KUKA KRL program: MyProgram_302().src

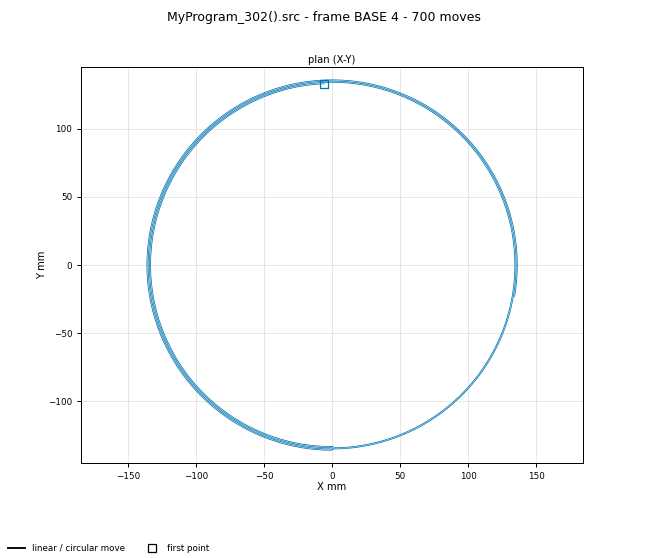
[picture p0: tool path of MyProgram_302().src in frame BASE 4, 700 of 700 moves have a stored position in this frame; points joined in program order, loops and branches not executed]
&ACCESS RVP
&REL 1
&PARAM TEMPLATE = C:\KRC\Roboter\Template\vorgabe
&PARAM EDITMASK = *
DEF MyProgram_302()
; ---- Setting reference (Base) ----
$BASE = BASE_DATA[4]

; --------------------------
; ---- Setting tool (TCP) ----
$TOOL = TOOL_DATA[3]
; --------------------------

$VEL.CP = VEL_APROX_PRINT
Startdeposition()
$VEL.CP = VEL_PRINT
LIN {X -5.8401,Y 133.2502,Z 180,A 93.9157,B 5.8389,C 0.0819,E1 5.8328,E2 358.4356} C_DIS
LIN {X -9.9087,Y 133.0081,Z 180,A 95.4392,B 5.8389,C 0.0849,E1 5.8286,E2 356.9401} C_DIS
LIN {X -13.164,Y 132.726,Z 180,A 96.8413,B 5.8389,C 0.0853,E1 5.8247,E2 355.5388} C_DIS
LIN {X -16.4317,Y 132.362,Z 180,A 98.2546,B 5.8389,C 0.0857,E1 5.8208,E2 354.1262} C_DIS
LIN {X -19.569,Y 131.9349,Z 180,A 99.6594,B 5.8389,C 0.0857,E1 5.8169,E2 352.7169} C_DIS
LIN {X -22.7973,Y 131.4155,Z 180,A 101.1451,B 5.8389,C 0.0853,E1 5.8128,E2 351.2223} C_DIS
LIN {X -26.0144,Y 130.8161,Z 180,A 102.4928,B 5.8389,C 0.0867,E1 5.8091,E2 349.8823} C_DIS
LIN {X -29.8878,Y 129.9846,Z 180,A 104.0027,B 5.8389,C 0.0899,E1 5.805,E2 348.3962} C_DIS
LIN {X -32.4071,Y 129.38,Z 180,A 105.3169,B 5.8389,C 0.0884,E1 5.8014,E2 347.0588} C_DIS
LIN {X -35.6706,Y 128.5181,Z 180,A 106.7192,B 5.8389,C 0.09,E1 5.7976,E2 345.663} C_DIS
LIN {X -39.0431,Y 127.5337,Z 180,A 108.1859,B 5.8388,C 0.0916,E1 5.7937,E2 344.2024} C_DIS
LIN {X -41.9497,Y 126.6076,Z 180,A 109.7012,B 5.8388,C 0.0904,E1 5.7896,E2 342.6636} C_DIS
LIN {X -46.4559,Y 125.0247,Z 180,A 111.6781,B 5.8388,C 0.0932,E1 5.7845,E2 340.697} C_DIS
LIN {X -49.6202,Y 123.8026,Z 180,A 113.0937,B 5.8388,C 0.0952,E1 5.7808,E2 339.2873} C_DIS
LIN {X -52.5449,Y 122.5903,Z 180,A 114.5896,B 5.8388,C 0.0952,E1 5.7769,E2 337.7762} C_DIS
LIN {X -55.543,Y 121.2616,Z 180,A 115.9158,B 5.8387,C 0.0977,E1 5.7736,E2 336.4609} C_DIS
LIN {X -58.4989,Y 119.864,Z 180,A 117.3346,B 5.8387,C 0.0992,E1 5.77,E2 335.0414} C_DIS
LIN {X -61.4202,Y 118.3941,Z 180,A 118.7379,B 5.8387,C 0.101,E1 5.7665,E2 333.6394} C_DIS
LIN {X -64.3234,Y 116.8431,Z 180,A 120.1855,B 5.8387,C 0.1026,E1 5.7629,E2 332.1889} C_DIS
LIN {X -67.1606,Y 115.2359,Z 180,A 121.6276,B 5.8386,C 0.1041,E1 5.7594,E2 330.743} C_DIS
LIN {X -69.9578,Y 113.5592,Z 180,A 123.0324,B 5.8386,C 0.1061,E1 5.7561,E2 329.3388} C_DIS
LIN {X -72.7953,Y 111.7614,Z 180,A 124.4937,B 5.8386,C 0.1081,E1 5.7527,E2 327.8763} C_DIS
LIN {X -75.4227,Y 110.0052,Z 180,A 125.8852,B 5.8385,C 0.1099,E1 5.7494,E2 326.4819} C_DIS
LIN {X -78.448,Y 107.8688,Z 180,A 127.5592,B 5.8385,C 0.1117,E1 5.7456,E2 324.7993} C_DIS
LIN {X -81.4564,Y 105.6156,Z 180,A 129.1159,B 5.8384,C 0.115,E1 5.7422,E2 323.2508} C_DIS
LIN {X -84.6152,Y 103.1022,Z 180,A 130.8894,B 5.8384,C 0.1177,E1 5.7383,E2 321.4741} C_DIS
LIN {X -87.1187,Y 100.9953,Z 180,A 132.463,B 5.8384,C 0.1186,E1 5.7349,E2 319.8816} C_DIS
LIN {X -90.2118,Y 98.2422,Z 180,A 134.2565,B 5.8382,C 0.1219,E1 5.7312,E2 318.0878} C_DIS
LIN {X -93.1509,Y 95.4606,Z 180,A 135.898,B 5.8382,C 0.1263,E1 5.7279,E2 316.4594} C_DIS
LIN {X -95.9962,Y 92.5986,Z 180,A 137.6763,B 5.8381,C 0.1293,E1 5.7245,E2 314.6773} C_DIS
LIN {X -98.8242,Y 89.574,Z 180,A 139.4792,B 5.838,C 0.1328,E1 5.721,E2 312.8731} C_DIS
LIN {X -101.5295,Y 86.4956,Z 180,A 141.4063,B 5.838,C 0.135,E1 5.7175,E2 310.9275} C_DIS
LIN {X -104.1336,Y 83.3429,Z 180,A 143.0495,B 5.8378,C 0.14,E1 5.7146,E2 309.2994} C_DIS
LIN {X -106.2103,Y 80.6799,Z 180,A 144.5409,B 5.8378,C 0.1428,E1 5.7121,E2 307.8044} C_DIS
LIN {X -108.0959,Y 78.1346,Z 180,A 145.9441,B 5.8377,C 0.1456,E1 5.7097,E2 306.3974} C_DIS
LIN {X -109.9841,Y 75.4533,Z 180,A 147.4489,B 5.8377,C 0.1479,E1 5.7073,E2 304.8823} C_DIS
LIN {X -111.8695,Y 72.6287,Z 180,A 148.8508,B 5.8375,C 0.152,E1 5.7052,E2 303.4885} C_DIS
LIN {X -113.5591,Y 69.9579,Z 180,A 150.2623,B 5.8375,C 0.1547,E1 5.7031,E2 302.0717} C_DIS
LIN {X -115.5146,Y 66.6793,Z 180,A 151.8127,B 5.8373,C 0.1596,E1 5.7009,E2 300.5336} C_DIS
LIN {X -116.8988,Y 64.2227,Z 180,A 153.1553,B 5.8373,C 0.1614,E1 5.6991,E2 299.1763} C_DIS
LIN {X -118.436,Y 61.3404,Z 180,A 154.5977,B 5.8372,C 0.1646,E1 5.6972,E2 297.7304} C_DIS
LIN {X -120.0778,Y 58.0592,Z 180,A 156.1261,B 5.8371,C 0.1691,E1 5.6953,E2 296.2091} C_DIS
LIN {X -121.3072,Y 55.4444,Z 180,A 157.4767,B 5.837,C 0.1713,E1 5.6937,E2 294.8465} C_DIS
LIN {X -122.9165,Y 51.7774,Z 180,A 159.3933,B 5.837,C 0.1739,E1 5.6916,E2 292.9078} C_DIS
LIN {X -124.4775,Y 47.9035,Z 180,A 161.1621,B 5.8368,C 0.179,E1 5.6898,E2 291.1436} C_DIS
LIN {X -126.0894,Y 43.4824,Z 180,A 163.1672,B 5.8366,C 0.1846,E1 5.6879,E2 289.1423} C_DIS
LIN {X -127.3112,Y 39.7702,Z 180,A 164.8428,B 5.8364,C 0.1892,E1 5.6865,E2 287.4686} C_DIS
LIN {X -128.0982,Y 37.151,Z 180,A 166.0629,B 5.8364,C 0.192,E1 5.6855,E2 286.244} C_DIS
LIN {X -128.9966,Y 33.9018,Z 180,A 167.5452,B 5.8362,C 0.1956,E1 5.6844,E2 284.7589} C_DIS
LIN {X -129.9243,Y 30.1519,Z 180,A 169.1106,B 5.8361,C 0.2011,E1 5.6834,E2 283.2062} C_DIS
LIN {X -130.5092,Y 27.5138,Z 180,A 170.4318,B 5.836,C 0.2029,E1 5.6826,E2 281.8666} C_DIS
LIN {X -131.1453,Y 24.3049,Z 180,A 171.8683,B 5.8359,C 0.2065,E1 5.6819,E2 280.4276} C_DIS
LIN {X -131.7018,Y 21.0799,Z 180,A 173.2973,B 5.8357,C 0.2103,E1 5.6812,E2 278.9969} C_DIS
LIN {X -132.1649,Y 17.947,Z 180,A 174.7293,B 5.8357,C 0.2135,E1 5.6807,E2 277.5573} C_DIS
LIN {X -132.5646,Y 14.7006,Z 180,A 176.1681,B 5.8355,C 0.2172,E1 5.6802,E2 276.1157} C_DIS
LIN {X -132.8853,Y 11.4385,Z 180,A 177.6287,B 5.8353,C 0.2207,E1 5.6798,E2 274.6498} C_DIS
LIN {X -133.1258,Y 8.1746,Z 180,A 179.0576,B 5.8353,C 0.2245,E1 5.6796,E2 273.2192} C_DIS
LIN {X -133.2866,Y 4.9068,Z 180,A -179.5165,B 5.8351,C 0.2283,E1 5.6794,E2 271.792} C_DIS
LIN {X -133.3749,Y 0.8313,Z 180,A -178.0632,B 5.8347,C 0.236,E1 5.6794,E2 270.3762} C_DIS
LIN {X -133.3679,Y -1.6325,Z 180,A -176.5813,B 5.8347,C 0.2352,E1 5.6794,E2 268.8437} C_DIS
LIN {X -133.2864,Y -4.9122,Z 180,A -175.1553,B 5.8347,C 0.239,E1 5.6794,E2 267.4167} C_DIS
LIN {X -133.1254,Y -8.1812,Z 180,A -173.7271,B 5.8345,C 0.2428,E1 5.6797,E2 265.9869} C_DIS
LIN {X -132.8762,Y -11.5458,Z 180,A -172.2661,B 5.8343,C 0.2468,E1 5.68,E2 264.5255} C_DIS
LIN {X -132.5536,Y -14.8028,Z 180,A -170.698,B 5.8342,C 0.2493,E1 5.6805,E2 262.9387} C_DIS
LIN {X -132.1502,Y -18.0593,Z 180,A -169.3858,B 5.834,C 0.2542,E1 5.681,E2 261.6395} C_DIS
LIN {X -131.6677,Y -21.2918,Z 180,A -167.9555,B 5.8338,C 0.2579,E1 5.6816,E2 260.2068} C_DIS
LIN {X -131.1247,Y -24.4125,Z 180,A -166.5253,B 5.8337,C 0.261,E1 5.6823,E2 258.7691} C_DIS
LIN {X -130.4641,Y -27.7227,Z 180,A -165.0366,B 5.8335,C 0.2647,E1 5.6831,E2 257.2766} C_DIS
LIN {X -129.7641,Y -30.8334,Z 180,A -163.6416,B 5.8334,C 0.2682,E1 5.684,E2 255.8794} C_DIS
LIN {X -128.9428,Y -34.1037,Z 180,A -162.1588,B 5.8332,C 0.2719,E1 5.6851,E2 254.3933} C_DIS
LIN {X -128.0976,Y -37.153,Z 180,A -160.7666,B 5.833,C 0.2753,E1 5.6861,E2 252.9979} C_DIS
LIN {X -127.1483,Y -40.2817,Z 180,A -159.3021,B 5.8329,C 0.2785,E1 5.6873,E2 251.5269} C_DIS
LIN {X -126.0624,Y -43.5603,Z 180,A -157.8574,B 5.8327,C 0.2829,E1 5.6886,E2 250.0879} C_DIS
LIN {X -125.0212,Y -46.4651,Z 180,A -156.4263,B 5.8326,C 0.2854,E1 5.69,E2 248.6445} C_DIS
LIN {X -123.5796,Y -50.1735,Z 180,A -154.8472,B 5.8323,C 0.2911,E1 5.6916,E2 247.0824} C_DIS
LIN {X -122.5879,Y -52.5505,Z 180,A -153.5732,B 5.8323,C 0.2924,E1 5.693,E2 245.7883} C_DIS
LIN {X -121.2627,Y -55.5407,Z 180,A -152.137,B 5.832,C 0.2957,E1 5.6947,E2 244.3491} C_DIS
LIN {X -119.838,Y -58.5516,Z 180,A -150.6937,B 5.8319,C 0.2992,E1 5.6964,E2 242.905} C_DIS
LIN {X -118.3945,Y -61.4194,Z 180,A -149.2856,B 5.8317,C 0.3023,E1 5.6982,E2 241.494} C_DIS
LIN {X -116.863,Y -64.2876,Z 180,A -147.8375,B 5.8315,C 0.3053,E1 5.7001,E2 240.0402} C_DIS
LIN {X -115.2646,Y -67.111,Z 180,A -146.2707,B 5.8315,C 0.307,E1 5.7024,E2 238.4526} C_DIS
LIN {X -113.5511,Y -69.9709,Z 180,A -144.9407,B 5.8312,C 0.3114,E1 5.7043,E2 237.136} C_DIS
LIN {X -111.7443,Y -72.8215,Z 180,A -143.4608,B 5.8311,C 0.3145,E1 5.7065,E2 235.6528} C_DIS
LIN {X -109.9836,Y -75.454,Z 180,A -142.0556,B 5.8309,C 0.3172,E1 5.7087,E2 234.2427} C_DIS
LIN {X -108.0943,Y -78.1368,Z 180,A -140.6414,B 5.8307,C 0.3204,E1 5.711,E2 232.8285} C_DIS
LIN {X -106.1145,Y -80.8053,Z 180,A -139.1884,B 5.8306,C 0.3233,E1 5.7135,E2 231.3728} C_DIS
LIN {X -103.6547,Y -83.9373,Z 180,A -137.4174,B 5.8304,C 0.3264,E1 5.7166,E2 229.5948} C_DIS
LIN {X -100.9949,Y -87.1191,Z 180,A -135.4726,B 5.8303,C 0.3284,E1 5.7201,E2 227.6303} C_DIS
LIN {X -98.237,Y -90.2175,Z 180,A -133.676,B 5.8301,C 0.3319,E1 5.7235,E2 225.8323} C_DIS
LIN {X -95.4637,Y -93.1478,Z 180,A -132.0371,B 5.8298,C 0.3364,E1 5.7266,E2 224.2056} C_DIS
LIN {X -92.6027,Y -95.9922,Z 180,A -130.2614,B 5.8297,C 0.3393,E1 5.7302,E2 222.4249} C_DIS
LIN {X -89.5801,Y -98.8186,Z 180,A -128.4607,B 5.8295,C 0.3423,E1 5.7339,E2 220.6216} C_DIS
LIN {X -86.4961,Y -101.529,Z 180,A -126.5401,B 5.8295,C 0.3438,E1 5.738,E2 218.6818} C_DIS
LIN {X -83.3456,Y -104.1314,Z 180,A -124.8384,B 5.8292,C 0.3474,E1 5.7417,E2 216.987} C_DIS
LIN {X -80.6705,Y -106.2174,Z 180,A -123.4167,B 5.829,C 0.3502,E1 5.7448,E2 215.5699} C_DIS
LIN {X -78.1287,Y -108.1002,Z 180,A -122.0232,B 5.829,C 0.352,E1 5.7479,E2 214.1722} C_DIS
LIN {X -75.4533,Y -109.9841,Z 180,A -120.618,B 5.8288,C 0.3541,E1 5.7512,E2 212.7671} C_DIS
LIN {X -72.6468,Y -111.8578,Z 180,A -119.1506,B 5.8287,C 0.3561,E1 5.7546,E2 211.2976} C_DIS
LIN {X -69.971,Y -113.551,Z 180,A -117.7497,B 5.8286,C 0.3575,E1 5.7579,E2 209.8917} C_DIS
LIN {X -67.0769,Y -115.2843,Z 180,A -116.2249,B 5.8286,C 0.3586,E1 5.7616,E2 208.3573} C_DIS
LIN {X -63.6192,Y -117.228,Z 180,A -114.6815,B 5.8283,C 0.3626,E1 5.7653,E2 206.834} C_DIS
LIN {X -61.3282,Y -118.4424,Z 180,A -113.4475,B 5.8283,C 0.3626,E1 5.7684,E2 205.5849} C_DIS
LIN {X -58.4051,Y -119.9102,Z 180,A -112.0301,B 5.8282,C 0.3641,E1 5.772,E2 204.1659} C_DIS
LIN {X -55.4488,Y -121.3052,Z 180,A -110.6141,B 5.8281,C 0.3655,E1 5.7756,E2 202.7482} C_DIS
LIN {X -52.4577,Y -122.6281,Z 180,A -109.206,B 5.8281,C 0.3669,E1 5.7792,E2 201.3396} C_DIS
LIN {X -49.5299,Y -123.839,Z 180,A -107.8163,B 5.8279,C 0.3679,E1 5.7828,E2 199.946} C_DIS
LIN {X -46.3584,Y -125.0612,Z 180,A -106.3358,B 5.8279,C 0.369,E1 5.7867,E2 198.4628} C_DIS
LIN {X -43.3991,Y -126.1182,Z 180,A -104.9873,B 5.8279,C 0.3701,E1 5.7902,E2 197.1142} C_DIS
LIN {X -40.2328,Y -127.1639,Z 180,A -103.5591,B 5.8277,C 0.3713,E1 5.794,E2 195.6862} C_DIS
LIN {X -37.2598,Y -128.0663,Z 180,A -102.1668,B 5.8277,C 0.3715,E1 5.7978,E2 194.2864} C_DIS
LIN {X -33.7056,Y -129.0489,Z 180,A -100.63,B 5.8277,C 0.3731,E1 5.8019,E2 192.7552} C_DIS
LIN {X -30.8137,Y -129.7689,Z 180,A -99.337,B 5.8276,C 0.3736,E1 5.8054,E2 191.4602} C_DIS
LIN {X -27.5186,Y -130.5082,Z 180,A -97.8837,B 5.8276,C 0.3743,E1 5.8094,E2 190.0062} C_DIS
LIN {X -24.3131,Y -131.1437,Z 180,A -96.3211,B 5.8276,C 0.3729,E1 5.8137,E2 188.4231} C_DIS
LIN {X -21.0911,Y -131.7001,Z 180,A -95.0816,B 5.8275,C 0.3754,E1 5.8171,E2 187.2041} C_DIS
LIN {X -17.958,Y -132.1635,Z 180,A -93.6817,B 5.8275,C 0.3754,E1 5.821,E2 185.7987} C_DIS
LIN {X -14.6983,Y -132.5648,Z 180,A -92.2718,B 5.8275,C 0.3756,E1 5.8249,E2 184.3883} C_DIS
LIN {X -11.4444,Y -132.8848,Z 180,A -90.8248,B 5.8275,C 0.3753,E1 5.8289,E2 182.9354} C_DIS
LIN {X -8.1833,Y -133.1253,Z 180,A -89.4562,B 5.8275,C 0.3758,E1 5.8327,E2 181.5708} C_DIS
LIN {X -4.9184,Y -133.2862,Z 180,A -88.0669,B 5.8275,C 0.376,E1 5.8366,E2 180.1828} C_DIS
LIN {X -1.6521,Y -133.3676,Z 180,A -86.6466,B 5.8275,C 0.3757,E1 5.8406,E2 178.7597} C_DIS
LIN {X 0.9654,Y -133.3724,Z 180,A -85.8773,B 5.8272,C 0.3801,E1 5.8426,E2 178.0345} C_DIS
Enddeposition()
LIN {X 0.9654,Y -133.3724,Z 180,A -85.8773,B 5.8272,C 0.3801,E1 5.8426,E2 178.0345} C_DIS
Startdeposition()
$VEL.CP = VEL_PRINT
LIN {X -1.8229,Y -134.2676,Z 180,A -87.4081,B 5.8265,C 0.3879,E1 5.838,E2 179.6414} C_DIS
LIN {X -5.9362,Y -134.1498,Z 180,A -89.2358,B 5.8265,C 0.3889,E1 5.8329,E2 181.479} C_DIS
LIN {X -10.4243,Y -133.8756,Z 180,A -90.9726,B 5.8266,C 0.3865,E1 5.8281,E2 183.1938} C_DIS
LIN {X -13.6518,Y -133.5853,Z 180,A -92.7112,B 5.8264,C 0.3907,E1 5.8232,E2 184.9776} C_DIS
LIN {X -16.9255,Y -133.2092,Z 180,A -93.6954,B 5.8267,C 0.3851,E1 5.8206,E2 185.9093} C_DIS
LIN {X -19.5444,Y -132.8503,Z 180,A -94.891,B 5.8267,C 0.3857,E1 5.8173,E2 187.1138} C_DIS
LIN {X -23.1124,Y -132.2762,Z 180,A -96.6307,B 5.8266,C 0.3876,E1 5.8124,E2 188.8789} C_DIS
LIN {X -27.0527,Y -131.526,Z 180,A -98.1959,B 5.8267,C 0.385,E1 5.8081,E2 190.4262} C_DIS
LIN {X -30.9558,Y -130.6631,Z 180,A -100.0353,B 5.8267,C 0.3858,E1 5.8031,E2 192.283} C_DIS
LIN {X -35.3302,Y -129.5499,Z 180,A -102.2882,B 5.8265,C 0.3885,E1 5.7969,E2 194.5771} C_DIS
LIN {X -39.0512,Y -128.4753,Z 180,A -103.9879,B 5.8265,C 0.3878,E1 5.7923,E2 196.283} C_DIS
LIN {X -43.1127,Y -127.171,Z 180,A -105.3156,B 5.827,C 0.3806,E1 5.789,E2 197.5496} C_DIS
LIN {X -46.1895,Y -126.0865,Z 180,A -107.0216,B 5.8269,C 0.3831,E1 5.7844,E2 199.2952} C_DIS
LIN {X -51.1313,Y -124.1645,Z 180,A -108.9572,B 5.8273,C 0.3772,E1 5.7795,E2 201.1902} C_DIS
LIN {X -53.5217,Y -123.1514,Z 180,A -110.1581,B 5.8273,C 0.3772,E1 5.7764,E2 202.4028} C_DIS
LIN {X -57.232,Y -121.4734,Z 180,A -111.8503,B 5.8274,C 0.3747,E1 5.7721,E2 204.0896} C_DIS
LIN {X -59.6757,Y -120.29,Z 180,A -113.1398,B 5.8274,C 0.3749,E1 5.7688,E2 205.3955} C_DIS
LIN {X -63.8676,Y -118.1202,Z 180,A -115.1667,B 5.8275,C 0.3725,E1 5.7638,E2 207.4242} C_DIS
LIN {X -67.6152,Y -116.0158,Z 180,A -117.0786,B 5.8276,C 0.371,E1 5.7591,E2 209.3458} C_DIS
LIN {X -70.8161,Y -114.0895,Z 180,A -118.5521,B 5.8279,C 0.3674,E1 5.7557,E2 210.8042} C_DIS
LIN {X -73.4828,Y -112.3912,Z 180,A -120.0772,B 5.8279,C 0.3674,E1 5.752,E2 212.3513} C_DIS
LIN {X -76.8332,Y -110.1272,Z 180,A -121.8054,B 5.828,C 0.3648,E1 5.7481,E2 214.0797} C_DIS
LIN {X -80.357,Y -107.583,Z 180,A -123.6442,B 5.8282,C 0.3617,E1 5.7439,E2 215.9164} C_DIS
LIN {X -83.8659,Y -104.871,Z 180,A -125.5135,B 5.8284,C 0.3583,E1 5.7398,E2 217.7826} C_DIS
LIN {X -86.7787,Y -102.4735,Z 180,A -127.2167,B 5.8286,C 0.3565,E1 5.7361,E2 219.4972} C_DIS
LIN {X -90.0905,Y -99.5744,Z 180,A -129.1455,B 5.8287,C 0.3536,E1 5.7321,E2 221.4319} C_DIS
LIN {X -93.5149,Y -96.3655,Z 180,A -131.098,B 5.829,C 0.3493,E1 5.7282,E2 223.3779} C_DIS
LIN {X -96.2125,Y -93.6729,Z 180,A -132.7735,B 5.8291,C 0.3466,E1 5.7249,E2 225.0592} C_DIS
LIN {X -98.7892,Y -90.9507,Z 180,A -134.4306,B 5.8293,C 0.344,E1 5.7217,E2 226.7229} C_DIS
LIN {X -101.2522,Y -88.2004,Z 180,A -136.0603,B 5.8295,C 0.3413,E1 5.7187,E2 228.359} C_DIS
LIN {X -104.2235,Y -84.6695,Z 180,A -138.0297,B 5.8297,C 0.3371,E1 5.7152,E2 230.3278} C_DIS
LIN {X -106.5852,Y -81.6757,Z 180,A -139.6703,B 5.8299,C 0.3336,E1 5.7124,E2 231.9695} C_DIS
LIN {X -109.0027,Y -78.4212,Z 180,A -141.522,B 5.83,C 0.331,E1 5.7093,E2 233.8356} C_DIS
LIN {X -111.7464,Y -74.4585,Z 180,A -143.4191,B 5.8304,C 0.3246,E1 5.7063,E2 235.7122} C_DIS
LIN {X -113.3521,Y -71.9914,Z 180,A -144.7748,B 5.8305,C 0.3227,E1 5.7043,E2 237.0798} C_DIS
LIN {X -115.3599,Y -68.7271,Z 180,A -147.8317,B 5.83,C 0.3326,E1 5.6997,E2 240.3093} C_DIS
LIN {X -119.6052,Y -61.0359,Z 180,A -149.9919,B 5.8313,C 0.3079,E1 5.6971,E2 242.274} C_DIS
LIN {X -121.4935,Y -57.19,Z 180,A -152.1421,B 5.8313,C 0.3064,E1 5.6944,E2 244.4631} C_DIS
LIN {X -122.6668,Y -54.6231,Z 180,A -153.3886,B 5.8315,C 0.3037,E1 5.693,E2 245.714} C_DIS
LIN {X -124.129,Y -51.2163,Z 180,A -154.9876,B 5.8317,C 0.2998,E1 5.6913,E2 247.3143} C_DIS
LIN {X -125.6383,Y -47.391,Z 180,A -156.5791,B 5.832,C 0.2936,E1 5.6897,E2 248.8847} C_DIS
LIN {X -126.422,Y -45.2589,Z 180,A -157.8208,B 5.832,C 0.2936,E1 5.6885,E2 250.1594} C_DIS
LIN {X -127.5238,Y -42.0553,Z 180,A -159.2082,B 5.8323,C 0.2892,E1 5.6872,E2 251.5388} C_DIS
LIN {X -128.5924,Y -38.6682,Z 180,A -160.7647,B 5.8324,C 0.2855,E1 5.6859,E2 253.0994} C_DIS
LIN {X -129.5062,Y -35.489,Z 180,A -162.3212,B 5.8326,C 0.283,E1 5.6848,E2 254.6729} C_DIS
LIN {X -130.9359,Y -29.7766,Z 180,A -164.7998,B 5.8329,C 0.2758,E1 5.6831,E2 257.1456} C_DIS
LIN {X -131.6865,Y -26.2638,Z 180,A -166.4132,B 5.8331,C 0.2723,E1 5.6822,E2 258.7678} C_DIS
LIN {X -132.284,Y -23.0684,Z 180,A -167.924,B 5.8331,C 0.2696,E1 5.6814,E2 260.2928} C_DIS
LIN {X -132.9526,Y -18.8284,Z 180,A -169.7276,B 5.8334,C 0.2642,E1 5.6807,E2 262.0917} C_DIS
LIN {X -133.4808,Y -14.6235,Z 180,A -171.5757,B 5.8337,C 0.2594,E1 5.6801,E2 263.9434} C_DIS
LIN {X -133.877,Y -10.4048,Z 180,A -173.3775,B 5.8339,C 0.2542,E1 5.6796,E2 265.7431} C_DIS
LIN {X -134.0726,Y -7.4837,Z 180,A -174.8802,B 5.8339,C 0.253,E1 5.6794,E2 267.2757} C_DIS
LIN {X -134.2477,Y -3.004,Z 180,A -176.7939,B 5.8342,C 0.2476,E1 5.6792,E2 269.188} C_DIS
LIN {X -134.2747,Y 1.2521,Z 180,A -178.5999,B 5.8344,C 0.2423,E1 5.6792,E2 270.9914} C_DIS
LIN {X -134.1737,Y 5.3251,Z 180,A 179.6874,B 5.8346,C 0.2371,E1 5.6794,E2 272.6995} C_DIS
LIN {X -134.0112,Y 8.4826,Z 180,A 178.3108,B 5.8347,C 0.2335,E1 5.6796,E2 274.0783} C_DIS
LIN {X -133.7853,Y 11.5076,Z 180,A 176.9868,B 5.8349,C 0.2301,E1 5.6799,E2 275.4049} C_DIS
LIN {X -133.4736,Y 14.6901,Z 180,A 175.5902,B 5.835,C 0.2265,E1 5.6803,E2 276.8043} C_DIS
LIN {X -133.0711,Y 17.9794,Z 180,A 173.9883,B 5.8351,C 0.2242,E1 5.6809,E2 278.4277} C_DIS
LIN {X -132.3686,Y 22.5758,Z 180,A 171.9674,B 5.8353,C 0.219,E1 5.6818,E2 280.4514} C_DIS
LIN {X -131.5306,Y 27.0302,Z 180,A 170.0654,B 5.8355,C 0.2133,E1 5.6828,E2 282.3479} C_DIS
LIN {X -130.446,Y 31.8568,Z 180,A 168.0066,B 5.8358,C 0.2069,E1 5.6841,E2 284.3986} C_DIS
LIN {X -129.6981,Y 34.7746,Z 180,A 166.5489,B 5.8358,C 0.2049,E1 5.6851,E2 285.876} C_DIS
LIN {X -128.7451,Y 38.154,Z 180,A 165.087,B 5.836,C 0.2005,E1 5.6863,E2 287.3322} C_DIS
LIN {X -127.7191,Y 41.4613,Z 180,A 163.6201,B 5.8361,C 0.1964,E1 5.6875,E2 288.7965} C_DIS
LIN {X -126.7327,Y 44.3825,Z 180,A 162.1143,B 5.8361,C 0.1946,E1 5.6889,E2 290.324} C_DIS
LIN {X -125.4252,Y 47.9571,Z 180,A 160.6153,B 5.8364,C 0.1891,E1 5.6904,E2 291.8066} C_DIS
LIN {X -124.4052,Y 50.5399,Z 180,A 159.3751,B 5.8364,C 0.1864,E1 5.6917,E2 293.0524} C_DIS
LIN {X -123.0342,Y 53.7929,Z 180,A 157.8355,B 5.8366,C 0.1828,E1 5.6933,E2 294.5946} C_DIS
LIN {X -121.6853,Y 56.7774,Z 180,A 156.378,B 5.8366,C 0.1797,E1 5.6951,E2 296.0582} C_DIS
LIN {X -119.6414,Y 60.9648,Z 180,A 154.5514,B 5.8368,C 0.1731,E1 5.6973,E2 297.8635} C_DIS
LIN {X -118.1614,Y 63.7909,Z 180,A 152.8627,B 5.8368,C 0.1728,E1 5.6995,E2 299.5904} C_DIS
LIN {X -116.0354,Y 67.5813,Z 180,A 150.9864,B 5.837,C 0.1684,E1 5.7021,E2 301.4677} C_DIS
LIN {X -114.1029,Y 70.7946,Z 180,A 148.9129,B 5.837,C 0.169,E1 5.7053,E2 303.596} C_DIS
LIN {X -111.7453,Y 74.4602,Z 180,A 147.4305,B 5.8372,C 0.1609,E1 5.7075,E2 305.0319} C_DIS
LIN {X -109.0975,Y 78.2886,Z 180,A 145.4013,B 5.8373,C 0.1567,E1 5.7107,E2 307.0645} C_DIS
LIN {X -106.8983,Y 81.2663,Z 180,A 143.8891,B 5.8374,C 0.1525,E1 5.7133,E2 308.5674} C_DIS
LIN {X -104.445,Y 84.3954,Z 180,A 142.0516,B 5.8374,C 0.1501,E1 5.7165,E2 310.4202} C_DIS
LIN {X -101.5169,Y 87.8963,Z 180,A 140.0565,B 5.8376,C 0.1463,E1 5.7201,E2 312.4191} C_DIS
LIN {X -98.5584,Y 91.2016,Z 180,A 138.1918,B 5.8376,C 0.142,E1 5.7236,E2 314.2789} C_DIS
LIN {X -95.7512,Y 94.1437,Z 180,A 136.3912,B 5.8378,C 0.1391,E1 5.7271,E2 316.0858} C_DIS
LIN {X -92.5547,Y 97.2884,Z 180,A 134.4713,B 5.8378,C 0.1354,E1 5.7309,E2 318.0048} C_DIS
LIN {X -89.2963,Y 100.2877,Z 180,A 132.5062,B 5.8379,C 0.1326,E1 5.735,E2 319.9773} C_DIS
LIN {X -85.941,Y 103.1776,Z 180,A 130.5766,B 5.8379,C 0.1295,E1 5.7391,E2 321.91} C_DIS
LIN {X -82.5668,Y 105.8971,Z 180,A 128.6761,B 5.838,C 0.1268,E1 5.7433,E2 323.8152} C_DIS
LIN {X -78.9123,Y 108.6471,Z 180,A 126.7683,B 5.8381,C 0.123,E1 5.7476,E2 325.7162} C_DIS
LIN {X -73.5343,Y 112.3573,Z 180,A 123.6484,B 5.8381,C 0.1221,E1 5.7549,E2 328.8731} C_DIS
LIN {X -70.5442,Y 114.2584,Z 180,A 122.6292,B 5.8383,C 0.1147,E1 5.7572,E2 329.8328} C_DIS
LIN {X -68.0549,Y 115.7577,Z 180,A 121.1966,B 5.8383,C 0.1149,E1 5.7607,E2 331.2873} C_DIS
LIN {X -63.1842,Y 118.4874,Z 180,A 118.804,B 5.8383,C 0.1118,E1 5.7665,E2 333.6794} C_DIS
LIN {X -59.0297,Y 120.6086,Z 180,A 116.7474,B 5.8383,C 0.11,E1 5.7717,E2 335.7422} C_DIS
LIN {X -56.1305,Y 121.9844,Z 180,A 115.4098,B 5.8384,C 0.108,E1 5.775,E2 337.0751} C_DIS
LIN {X -52.8449,Y 123.4441,Z 180,A 113.7464,B 5.8384,C 0.1077,E1 5.7793,E2 338.7528} C_DIS
LIN {X -49.6878,Y 124.7486,Z 180,A 111.4479,B 5.8383,C 0.1154,E1 5.7856,E2 341.1489} C_DIS
LIN {X -43.5256,Y 127.0298,Z 180,A 109.5502,B 5.8385,C 0.1028,E1 5.7903,E2 342.9385} C_DIS
LIN {X -38.0339,Y 128.7802,Z 180,A 107.2884,B 5.8385,C 0.0986,E1 5.7962,E2 345.1752} C_DIS
LIN {X -35.2972,Y 129.5587,Z 180,A 105.9102,B 5.8385,C 0.0995,E1 5.8,E2 346.5723} C_DIS
LIN {X -32.4186,Y 130.3084,Z 180,A 104.6358,B 5.8385,C 0.0987,E1 5.8034,E2 347.8465} C_DIS
LIN {X -29.6954,Y 130.9545,Z 180,A 103.3822,B 5.8385,C 0.0987,E1 5.8069,E2 349.1063} C_DIS
LIN {X -25.9469,Y 131.7504,Z 180,A 101.7804,B 5.8385,C 0.0974,E1 5.8112,E2 350.7033} C_DIS
LIN {X -22.9099,Y 132.3123,Z 180,A 100.292,B 5.8385,C 0.0988,E1 5.8154,E2 352.2111} C_DIS
LIN {X -18.4899,Y 133.001,Z 180,A 98.5148,B 5.8386,C 0.0965,E1 5.8202,E2 353.9718} C_DIS
LIN {X -13.0322,Y 133.6454,Z 180,A 96.3422,B 5.8386,C 0.0938,E1 5.8262,E2 356.1226} C_DIS
LIN {X -9.7194,Y 133.927,Z 180,A 94.6822,B 5.8386,C 0.0964,E1 5.8309,E2 357.8105} C_DIS
LIN {X -6.088,Y 134.1428,Z 180,A 93.0193,B 5.8386,C 0.0975,E1 5.8356,E2 359.4859} C_DIS
LIN {X -2.467,Y 134.2569,Z 180,A 91.5934,B 5.8386,C 0.096,E1 5.8395,E2 360.8969} C_DIS
LIN {X 1.1007,Y 134.2753,Z 180,A 90.1887,B 5.8386,C 0.0946,E1 5.8434,E2 362.2869} C_DIS
LIN {X 4.6564,Y 134.1998,Z 180,A 88.6949,B 5.8386,C 0.0945,E1 5.8476,E2 363.7774} C_DIS
LIN {X 7.3307,Y 134.0803,Z 180,A 87.2919,B 5.8386,C 0.0979,E1 5.8516,E2 365.2108} C_DIS
LIN {X 10.9211,Y 133.8349,Z 180,A 85.7758,B 5.8386,C 0.098,E1 5.8558,E2 366.724} C_DIS
LIN {X 14.8909,Y 133.452,Z 180,A 84.23,B 5.8386,C 0.0967,E1 5.86,E2 368.2507} C_DIS
LIN {X 18.887,Y 132.9442,Z 180,A 82.568,B 5.8386,C 0.0967,E1 5.8646,E2 369.9053} C_DIS
LIN {X 22.3354,Y 132.4087,Z 180,A 81.0552,B 5.8386,C 0.0977,E1 5.8688,E2 371.4205} C_DIS
LIN {X 25.9928,Y 131.7416,Z 180,A 79.3333,B 5.8386,C 0.1003,E1 5.8736,E2 373.1581} C_DIS
LIN {X 30.1267,Y 130.8559,Z 180,A 77.6008,B 5.8386,C 0.1005,E1 5.8783,E2 374.8816} C_DIS
LIN {X 35.9171,Y 129.3865,Z 180,A 74.6568,B 5.8384,C 0.1076,E1 5.8863,E2 377.8718} C_DIS
LIN {X 39.9713,Y 128.1932,Z 180,A 73.3449,B 5.8385,C 0.1027,E1 5.8897,E2 379.1251} C_DIS
LIN {X 43.235,Y 127.1305,Z 180,A 71.6493,B 5.8385,C 0.1071,E1 5.8942,E2 380.848} C_DIS
LIN {X 47.3091,Y 125.669,Z 180,A 69.9995,B 5.8385,C 0.1064,E1 5.8985,E2 382.4739} C_DIS
LIN {X 50.6514,Y 124.3602,Z 180,A 68.5478,B 5.8385,C 0.107,E1 5.9022,E2 383.916} C_DIS
LIN {X 53.9842,Y 122.9515,Z 180,A 67.0057,B 5.8384,C 0.1087,E1 5.9062,E2 385.4578} C_DIS
LIN {X 56.7098,Y 121.7166,Z 180,A 65.7474,B 5.8384,C 0.11,E1 5.9094,E2 386.7137} C_DIS
LIN {X 59.7538,Y 120.2514,Z 180,A 64.2889,B 5.8384,C 0.1121,E1 5.9131,E2 388.1741} C_DIS
LIN {X 63.6861,Y 118.2177,Z 180,A 62.356,B 5.8383,C 0.1152,E1 5.9178,E2 390.1123} C_DIS
LIN {X 67.593,Y 116.0286,Z 180,A 60.5146,B 5.8383,C 0.117,E1 5.9223,E2 391.9454} C_DIS
LIN {X 70.7099,Y 114.1556,Z 180,A 59.0352,B 5.8383,C 0.1184,E1 5.9258,E2 393.4163} C_DIS
LIN {X 73.8141,Y 112.1731,Z 180,A 57.4868,B 5.8382,C 0.1205,E1 5.9294,E2 394.9618} C_DIS
LIN {X 76.9618,Y 110.0377,Z 180,A 55.7717,B 5.8381,C 0.1244,E1 5.9334,E2 396.6881} C_DIS
LIN {X 80.1819,Y 107.7134,Z 180,A 54.1128,B 5.8381,C 0.1268,E1 5.9371,E2 398.3429} C_DIS
LIN {X 83.8198,Y 104.9076,Z 180,A 52.2256,B 5.838,C 0.1293,E1 5.9413,E2 400.2217} C_DIS
LIN {X 86.605,Y 102.6208,Z 180,A 50.6696,B 5.838,C 0.1323,E1 5.9446,E2 401.7801} C_DIS
LIN {X 90.4223,Y 99.2733,Z 180,A 48.7849,B 5.838,C 0.1324,E1 5.9485,E2 403.6314} C_DIS
LIN {X 92.5684,Y 97.2754,Z 180,A 47.3214,B 5.8378,C 0.1379,E1 5.9515,E2 405.1207} C_DIS
LIN {X 95.577,Y 94.3214,Z 180,A 45.5045,B 5.8377,C 0.1418,E1 5.9551,E2 406.9401} C_DIS
LIN {X 98.0657,Y 91.7307,Z 180,A 44.0118,B 5.8377,C 0.1445,E1 5.9579,E2 408.4283} C_DIS
LIN {X 101.1335,Y 88.3364,Z 180,A 42.1376,B 5.8375,C 0.1475,E1 5.9614,E2 410.2937} C_DIS
LIN {X 103.996,Y 84.9479,Z 180,A 40.2576,B 5.8375,C 0.1515,E1 5.9648,E2 412.1728} C_DIS
LIN {X 106.8095,Y 81.3825,Z 180,A 38.4037,B 5.8374,C 0.1546,E1 5.9679,E2 414.0172} C_DIS
LIN {X 109.4242,Y 77.8316,Z 180,A 36.5302,B 5.8373,C 0.1588,E1 5.971,E2 415.8904} C_DIS
LIN {X 111.8797,Y 74.2589,Z 180,A 34.6686,B 5.8371,C 0.1634,E1 5.9739,E2 417.7542} C_DIS
LIN {X 114.0626,Y 70.8594,Z 180,A 33.0981,B 5.8371,C 0.1652,E1 5.9762,E2 419.3068} C_DIS
LIN {X 116.1136,Y 67.4462,Z 180,A 31.3436,B 5.8369,C 0.1702,E1 5.9787,E2 421.0688} C_DIS
LIN {X 118.309,Y 63.5162,Z 180,A 29.3918,B 5.8368,C 0.1755,E1 5.9814,E2 423.0253} C_DIS
LIN {X 120.4073,Y 59.4379,Z 180,A 27.5615,B 5.8367,C 0.1786,E1 5.9836,E2 424.8411} C_DIS
LIN {X 122.1459,Y 55.7813,Z 180,A 25.9847,B 5.8367,C 0.1807,E1 5.9855,E2 426.4005} C_DIS
LIN {X 123.2458,Y 53.3035,Z 180,A 24.4653,B 5.8363,C 0.1893,E1 5.9872,E2 427.9644} C_DIS
LIN {X 124.6709,Y 49.8805,Z 180,A 22.7558,B 5.8361,C 0.1954,E1 5.989,E2 429.6902} C_DIS
LIN {X 126.2827,Y 45.6454,Z 180,A 21.2942,B 5.8362,C 0.1934,E1 5.9904,E2 431.0958} C_DIS
LIN {X 128.0814,Y 40.3271,Z 180,A 19.0623,B 5.8361,C 0.1974,E1 5.9923,E2 433.3092} C_DIS
LIN {X 129.2445,Y 36.4247,Z 180,A 17.3443,B 5.8359,C 0.2018,E1 5.9936,E2 435.0259} C_DIS
LIN {X 130.2613,Y 32.604,Z 180,A 15.5872,B 5.8357,C 0.2075,E1 5.9949,E2 436.7927} C_DIS
LIN {X 131.3604,Y 27.8488,Z 180,A 13.6961,B 5.8357,C 0.2104,E1 5.996,E2 438.6617} C_DIS
LIN {X 132.0168,Y 24.5537,Z 180,A 12.2804,B 5.8355,C 0.2141,E1 5.9968,E2 440.0762} C_DIS
LIN {X 132.6829,Y 20.6428,Z 180,A 10.6122,B 5.8353,C 0.2185,E1 5.9975,E2 441.7425} C_DIS
LIN {X 133.2533,Y 16.5799,Z 180,A 8.9812,B 5.8353,C 0.2216,E1 5.9981,E2 443.3602} C_DIS
LIN {X 133.5382,Y 14.0897,Z 180,A 7.943,B 5.8351,C 0.2241,E1 5.9984,E2 444.3953} C_DIS
LIN {X 133.7815,Y 11.5538,Z 180,A 6.9204,B 5.8351,C 0.2262,E1 5.9987,E2 445.4108} C_DIS
LIN {X 133.9836,Y 8.9309,Z 180,A 5.7832,B 5.8349,C 0.2296,E1 5.9989,E2 446.5507} C_DIS
LIN {X 134.1437,Y 6.0686,Z 180,A 4.3933,B 5.8347,C 0.2357,E1 5.9991,E2 447.962} C_DIS
LIN {X 134.2708,Y 1.6275,Z 180,A 2.7791,B 5.8347,C 0.2367,E1 5.9992,E2 449.543} C_DIS
LIN {X 134.278,Y -0.7661,Z 180,A 1.5874,B 5.8344,C 0.2423,E1 5.9992,E2 450.7565} C_DIS
LIN {X 134.1797,Y -5.1715,Z 180,A -0.2,B 5.8342,C 0.2462,E1 5.9991,E2 452.5339} C_DIS
LIN {X 133.9953,Y -8.7404,Z 180,A -1.7823,B 5.834,C 0.2515,E1 5.9988,E2 454.1246} C_DIS
LIN {X 133.7002,Y -12.4622,Z 180,A -3.0901,B 5.834,C 0.2515,E1 5.9985,E2 455.3985} C_DIS
LIN {X 133.4347,Y -15.0517,Z 180,A -4.2486,B 5.8338,C 0.2555,E1 5.9981,E2 456.5638} C_DIS
LIN {X 133.1148,Y -17.6456,Z 180,A -5.3021,B 5.8338,C 0.2577,E1 5.9978,E2 457.6105} C_DIS
LIN {X 132.7618,Y -20.1331,Z 180,A -6.3337,B 5.8336,C 0.2601,E1 5.9973,E2 458.6381} C_DIS
LIN {X 132.1676,Y -23.719,Z 180,A -8.0262,B 5.8333,C 0.2667,E1 5.9965,E2 460.3494} C_DIS
LIN {X 131.4342,Y -27.504,Z 180,A -9.5034,B 5.8333,C 0.2687,E1 5.9957,E2 461.8073} C_DIS
LIN {X 130.809,Y -30.3322,Z 180,A -10.7,B 5.8331,C 0.2715,E1 5.995,E2 463.0001} C_DIS
LIN {X 129.9833,Y -33.6994,Z 180,A -12.5818,B 5.8326,C 0.2819,E1 5.9937,E2 464.933} C_DIS
LIN {X 128.9879,Y -37.3245,Z 180,A -13.5942,B 5.8328,C 0.2772,E1 5.993,E2 465.8736} C_DIS
LIN {X 128.1469,Y -40.1223,Z 180,A -15.2321,B 5.8324,C 0.2867,E1 5.9916,E2 467.5611} C_DIS
LIN {X 126.787,Y -44.226,Z 180,A -16.7826,B 5.8324,C 0.2871,E1 5.9902,E2 469.0767} C_DIS
LIN {X 125.5875,Y -47.5267,Z 180,A -18.2485,B 5.8322,C 0.2907,E1 5.9888,E2 470.54} C_DIS
LIN {X 124.3801,Y -50.6021,Z 180,A -19.7542,B 5.8319,C 0.2959,E1 5.9872,E2 472.0588} C_DIS
LIN {X 122.8993,Y -54.1033,Z 180,A -21.1764,B 5.8319,C 0.2971,E1 5.9856,E2 473.4577} C_DIS
LIN {X 121.7994,Y -56.5308,Z 180,A -22.4118,B 5.8316,C 0.3016,E1 5.9842,E2 474.7063} C_DIS
LIN {X 120.1974,Y -59.8633,Z 180,A -23.9141,B 5.8315,C 0.3046,E1 5.9823,E2 476.2008} C_DIS
LIN {X 117.7723,Y -64.5063,Z 180,A -26.0771,B 5.8312,C 0.3092,E1 5.9795,E2 478.3568} C_DIS
LIN {X 115.7201,Y -68.119,Z 180,A -27.8288,B 5.831,C 0.3133,E1 5.9771,E2 480.1075} C_DIS
LIN {X 113.4985,Y -71.7594,Z 180,A -29.6084,B 5.8308,C 0.3172,E1 5.9745,E2 481.8837} C_DIS
LIN {X 111.089,Y -75.4359,Z 180,A -31.4124,B 5.8306,C 0.3207,E1 5.9717,E2 483.6805} C_DIS
LIN {X 108.7347,Y -78.7914,Z 180,A -33.1894,B 5.8304,C 0.3253,E1 5.9688,E2 485.4626} C_DIS
LIN {X 106.2386,Y -82.1262,Z 180,A -34.9484,B 5.8302,C 0.3291,E1 5.9658,E2 487.2209} C_DIS
LIN {X 103.4377,Y -85.6269,Z 180,A -36.7763,B 5.83,C 0.3322,E1 5.9626,E2 489.04} C_DIS
LIN {X 100.3101,Y -89.2713,Z 180,A -38.796,B 5.8297,C 0.3363,E1 5.9589,E2 491.0578} C_DIS
LIN {X 97.6698,Y -92.1517,Z 180,A -40.4063,B 5.8296,C 0.339,E1 5.9559,E2 492.6625} C_DIS
LIN {X 95.0154,Y -94.8868,Z 180,A -42.0921,B 5.8293,C 0.3433,E1 5.9525,E2 494.3571} C_DIS
LIN {X 90.9424,Y -98.7968,Z 180,A -44.4382,B 5.8291,C 0.3473,E1 5.9478,E2 496.6975} C_DIS
LIN {X 87.7085,Y -101.6786,Z 180,A -46.2026,B 5.829,C 0.3497,E1 5.9441,E2 498.453} C_DIS
LIN {X 84.6541,Y -104.2361,Z 180,A -47.8796,B 5.8288,C 0.3526,E1 5.9405,E2 500.1286} C_DIS
LIN {X 81.293,Y -106.8779,Z 180,A -49.7319,B 5.8286,C 0.3563,E1 5.9364,E2 501.986} C_DIS
LIN {X 78.3449,Y -109.0572,Z 180,A -51.1845,B 5.8285,C 0.3575,E1 5.9331,E2 503.4259} C_DIS
LIN {X 74.9335,Y -111.4291,Z 180,A -52.9597,B 5.8283,C 0.3605,E1 5.929,E2 505.2029} C_DIS
LIN {X 71.3424,Y -113.7618,Z 180,A -54.6695,B 5.8283,C 0.3618,E1 5.9251,E2 506.8995} C_DIS
LIN {X 68.885,Y -115.2658,Z 180,A -55.9225,B 5.8281,C 0.3641,E1 5.9221,E2 508.1564} C_DIS
LIN {X 65.418,Y -117.2689,Z 180,A -57.6919,B 5.8279,C 0.3675,E1 5.9177,E2 509.9348} C_DIS
LIN {X 61.4883,Y -119.3749,Z 180,A -59.405,B 5.8279,C 0.3675,E1 5.9136,E2 511.6256} C_DIS
LIN {X 58.5068,Y -120.8644,Z 180,A -60.8296,B 5.8277,C 0.3695,E1 5.91,E2 513.0516} C_DIS
LIN {X 55.3069,Y -122.361,Z 180,A -62.2588,B 5.8277,C 0.3704,E1 5.9064,E2 514.472} C_DIS
LIN {X 53.02,Y -123.3684,Z 180,A -64.0802,B 5.8269,C 0.3823,E1 5.9015,E2 516.3888} C_DIS
LIN {X 48.2363,Y -125.3166,Z 180,A -65.7499,B 5.8272,C 0.3774,E1 5.8973,E2 517.9934} C_DIS
LIN {X 42.2294,Y -127.4658,Z 180,A -68.3055,B 5.8272,C 0.378,E1 5.8906,E2 520.53} C_DIS
LIN {X 38.9799,Y -128.4971,Z 180,A -69.8346,B 5.827,C 0.3804,E1 5.8865,E2 522.0695} C_DIS
LIN {X 34.7041,Y -129.7169,Z 180,A -71.7411,B 5.827,C 0.3822,E1 5.8814,E2 523.9783} C_DIS
LIN {X 30.9329,Y -130.6687,Z 180,A -73.2707,B 5.827,C 0.3817,E1 5.8772,E2 525.4927} C_DIS
LIN {X 27.9883,Y -131.3302,Z 180,A -74.5948,B 5.8269,C 0.3831,E1 5.8736,E2 526.8222} C_DIS
LIN {X 23.1189,Y -132.275,Z 180,A -76.6087,B 5.8269,C 0.3831,E1 5.8681,E2 528.8245} C_DIS
LIN {X 19.7403,Y -132.8223,Z 180,A -78.3,B 5.8266,C 0.387,E1 5.8634,E2 530.5457} C_DIS
LIN {X 15.0256,Y -133.4375,Z 180,A -80.0749,B 5.8268,C 0.3846,E1 5.8585,E2 532.2898} C_DIS
LIN {X 11.7138,Y -133.7679,Z 180,A -81.8915,B 5.8264,C 0.3904,E1 5.8533,E2 534.157} C_DIS
LIN {X 8.3201,Y -134.0212,Z 180,A -83.0019,B 5.8267,C 0.3864,E1 5.8504,E2 535.2252} C_DIS
LIN {X 4.7775,Y -134.195,Z 180,A -84.4751,B 5.8267,C 0.3862,E1 5.8463,E2 536.6942} C_DIS
LIN {X 0.963,Y -134.2751,Z 180,A -86.3247,B 5.8265,C 0.3893,E1 5.841,E2 538.5723} C_DIS
Enddeposition()
LIN {X 0.963,Y -134.2751,Z 180,A -86.3247,B 5.8265,C 0.3893,E1 5.841,E2 538.5723} C_DIS
Startdeposition()
$VEL.CP = VEL_PRINT
LIN {X 1.5152,Y -135.1755,Z 180,A -85.1157,B 5.8271,C 0.38,E1 5.8447,E2 537.2721} C_DIS
LIN {X 8.0157,Y -134.9444,Z 180,A -82.393,B 5.8271,C 0.3797,E1 5.8523,E2 534.5525} C_DIS
LIN {X 14.4478,Y -134.4075,Z 180,A -79.7821,B 5.8271,C 0.3804,E1 5.8595,E2 531.9562} C_DIS
LIN {X 17.7195,Y -134.0155,Z 180,A -78.3412,B 5.8271,C 0.3791,E1 5.8635,E2 530.5088} C_DIS
LIN {X 21.6605,Y -133.4364,Z 180,A -76.4317,B 5.8274,C 0.3751,E1 5.8689,E2 528.5699} C_DIS
LIN {X 26.5456,Y -132.5504,Z 180,A -74.5835,B 5.8273,C 0.3773,E1 5.8738,E2 526.7533} C_DIS
LIN {X 29.6723,Y -131.8857,Z 180,A -73.1743,B 5.8273,C 0.3755,E1 5.8777,E2 525.3364} C_DIS
LIN {X 32.9894,Y -131.0948,Z 180,A -71.8122,B 5.8273,C 0.3755,E1 5.8814,E2 523.984} C_DIS
LIN {X 36.0021,Y -130.3,Z 180,A -70.4737,B 5.8275,C 0.3741,E1 5.885,E2 522.6423} C_DIS
LIN {X 39.4463,Y -129.2983,Z 180,A -69.0109,B 5.8275,C 0.3735,E1 5.8889,E2 521.1859} C_DIS
LIN {X 42.5226,Y -128.3196,Z 180,A -67.5838,B 5.8277,C 0.3713,E1 5.8927,E2 519.7502} C_DIS
LIN {X 46.7066,Y -126.8586,Z 180,A -65.6406,B 5.8278,C 0.3684,E1 5.8978,E2 517.7974} C_DIS
LIN {X 53.4902,Y -124.1485,Z 180,A -62.7267,B 5.8279,C 0.3673,E1 5.9053,E2 514.9047} C_DIS
LIN {X 56.4206,Y -122.8448,Z 180,A -61.2867,B 5.8281,C 0.3644,E1 5.909,E2 513.4533} C_DIS
LIN {X 59.6892,Y -121.2898,Z 180,A -59.7706,B 5.8281,C 0.3626,E1 5.9128,E2 511.9384} C_DIS
LIN {X 63.6651,Y -119.2537,Z 180,A -57.8919,B 5.8284,C 0.3601,E1 5.9175,E2 510.0601} C_DIS
LIN {X 67.3567,Y -117.2084,Z 180,A -56.0911,B 5.8285,C 0.3573,E1 5.9218,E2 508.2564} C_DIS
LIN {X 71.107,Y -114.9717,Z 180,A -54.2792,B 5.8287,C 0.3549,E1 5.9262,E2 506.448} C_DIS
LIN {X 74.6851,Y -112.6803,Z 180,A -52.4971,B 5.8288,C 0.3522,E1 5.9303,E2 504.6668} C_DIS
LIN {X 78.0581,Y -110.3699,Z 180,A -50.8536,B 5.8289,C 0.3505,E1 5.9341,E2 503.0333} C_DIS
LIN {X 81.54,Y -107.823,Z 180,A -49.0372,B 5.8291,C 0.3474,E1 5.9381,E2 501.2168} C_DIS
LIN {X 84.9391,Y -105.1661,Z 180,A -47.2326,B 5.8293,C 0.3444,E1 5.9421,E2 499.4137} C_DIS
LIN {X 88.4447,Y -102.2359,Z 180,A -45.3395,B 5.8295,C 0.3413,E1 5.9461,E2 497.5245} C_DIS
LIN {X 94.4708,Y -96.6948,Z 180,A -41.9082,B 5.8299,C 0.3349,E1 5.9531,E2 494.0952} C_DIS
LIN {X 97.6238,Y -93.5103,Z 180,A -40.0396,B 5.8301,C 0.3314,E1 5.9567,E2 492.2289} C_DIS
LIN {X 99.7419,Y -91.2481,Z 180,A -38.497,B 5.8304,C 0.325,E1 5.9597,E2 490.6558} C_DIS
LIN {X 102.1437,Y -88.5517,Z 180,A -37.2114,B 5.8304,C 0.3254,E1 5.962,E2 489.4002} C_DIS
LIN {X 104.9819,Y -85.1674,Z 180,A -35.4006,B 5.8306,C 0.3221,E1 5.9652,E2 487.5955} C_DIS
LIN {X 107.6411,Y -81.7809,Z 180,A -33.591,B 5.8308,C 0.3181,E1 5.9683,E2 485.7863} C_DIS
LIN {X 110.3113,Y -78.1411,Z 180,A -31.7392,B 5.831,C 0.3145,E1 5.9713,E2 483.9406} C_DIS
LIN {X 112.5118,Y -74.9377,Z 180,A -30.1877,B 5.8311,C 0.312,E1 5.9737,E2 482.3997} C_DIS
LIN {X 114.8174,Y -71.355,Z 180,A -28.4238,B 5.8313,C 0.3082,E1 5.9763,E2 480.6395} C_DIS
LIN {X 116.8867,Y -67.9124,Z 180,A -26.6835,B 5.8316,C 0.3034,E1 5.9788,E2 478.8929} C_DIS
LIN {X 118.645,Y -64.7915,Z 180,A -24.5723,B 5.8322,C 0.2902,E1 5.9818,E2 476.7045} C_DIS
LIN {X 121.2363,Y -59.7976,Z 180,A -23.0216,B 5.8319,C 0.2971,E1 5.9836,E2 475.2581} C_DIS
LIN {X 122.6538,Y -56.8337,Z 180,A -21.6676,B 5.832,C 0.2941,E1 5.9852,E2 473.9077} C_DIS
LIN {X 123.8189,Y -54.2524,Z 180,A -20.3963,B 5.8323,C 0.2898,E1 5.9866,E2 472.6264} C_DIS
LIN {X 125.2945,Y -50.7481,Z 180,A -18.4426,B 5.8327,C 0.2801,E1 5.9887,E2 470.6276} C_DIS
LIN {X 126.7679,Y -46.9486,Z 180,A -17.402,B 5.8324,C 0.2863,E1 5.9897,E2 469.6727} C_DIS
LIN {X 128.4316,Y -42.186,Z 180,A -14.9887,B 5.8329,C 0.2761,E1 5.9919,E2 467.2228} C_DIS
LIN {X 129.6104,Y -38.411,Z 180,A -13.557,B 5.8329,C 0.2754,E1 5.993,E2 465.8206} C_DIS
LIN {X 130.6264,Y -34.7966,Z 180,A -11.8365,B 5.8333,C 0.2689,E1 5.9943,E2 464.0823} C_DIS
LIN {X 131.708,Y -30.4501,Z 180,A -9.9904,B 5.8335,C 0.2645,E1 5.9955,E2 462.2412} C_DIS
LIN {X 132.4841,Y -26.8712,Z 180,A -8.499,B 5.8336,C 0.2611,E1 5.9963,E2 460.7561} C_DIS
LIN {X 133.6671,Y -20.1859,Z 180,A -5.7175,B 5.8339,C 0.2545,E1 5.9977,E2 457.9844} C_DIS
LIN {X 134.1871,Y -16.3728,Z 180,A -4.0741,B 5.8341,C 0.2496,E1 5.9982,E2 456.3381} C_DIS
LIN {X 134.6067,Y -12.4646,Z 180,A -2.5177,B 5.8342,C 0.2466,E1 5.9987,E2 454.7941} C_DIS
LIN {X 134.9465,Y -7.9809,Z 180,A -0.2812,B 5.8347,C 0.2359,E1 5.9991,E2 452.5144} C_DIS
LIN {X 135.1161,Y -4.2477,Z 180,A 0.792,B 5.8345,C 0.2396,E1 5.9991,E2 451.5042} C_DIS
LIN {X 135.1804,Y -0.8077,Z 180,A 2.2446,B 5.8347,C 0.2355,E1 5.9992,E2 450.0512} C_DIS
LIN {X 135.0704,Y 5.4956,Z 180,A 5.2177,B 5.8352,C 0.2231,E1 5.999,E2 447.0382} C_DIS
LIN {X 134.8941,Y 8.8321,Z 180,A 6.3057,B 5.8352,C 0.2242,E1 5.9988,E2 445.9904} C_DIS
LIN {X 134.6057,Y 12.4756,Z 180,A 7.8589,B 5.8353,C 0.2198,E1 5.9985,E2 444.4356} C_DIS
LIN {X 134.2383,Y 15.9438,Z 180,A 9.4219,B 5.8355,C 0.2142,E1 5.998,E2 442.8608} C_DIS
LIN {X 133.6182,Y 20.5019,Z 180,A 11.1513,B 5.8355,C 0.2122,E1 5.9973,E2 441.1576} C_DIS
LIN {X 133.0739,Y 23.7786,Z 180,A 12.4336,B 5.8357,C 0.2102,E1 5.9967,E2 439.89} C_DIS
LIN {X 132.4427,Y 27.0746,Z 180,A 13.9734,B 5.8359,C 0.2044,E1 5.9958,E2 438.3346} C_DIS
LIN {X 131.4964,Y 31.3508,Z 180,A 15.7672,B 5.836,C 0.2002,E1 5.9947,E2 436.5474} C_DIS
LIN {X 130.6847,Y 34.5782,Z 180,A 17.1927,B 5.8361,C 0.1961,E1 5.9937,E2 435.1192} C_DIS
LIN {X 129.6011,Y 38.4428,Z 180,A 18.8034,B 5.8363,C 0.1929,E1 5.9925,E2 433.5187} C_DIS
LIN {X 128.1026,Y 43.174,Z 180,A 20.9441,B 5.8365,C 0.1866,E1 5.9906,E2 431.3721} C_DIS
LIN {X 126.6934,Y 47.1477,Z 180,A 22.6434,B 5.8365,C 0.1832,E1 5.989,E2 429.6826} C_DIS
LIN {X 124.9514,Y 51.5895,Z 180,A 24.7871,B 5.8368,C 0.1759,E1 5.9868,E2 427.5227} C_DIS
LIN {X 122.9023,Y 56.2963,Z 180,A 26.7244,B 5.8368,C 0.174,E1 5.9846,E2 425.6139} C_DIS
LIN {X 121.3932,Y 59.4797,Z 180,A 28.1282,B 5.8369,C 0.1715,E1 5.9829,E2 424.2204} C_DIS
LIN {X 119.8145,Y 62.5985,Z 180,A 29.5787,B 5.837,C 0.1682,E1 5.981,E2 422.773} C_DIS
LIN {X 117.895,Y 66.1464,Z 180,A 31.3535,B 5.8372,C 0.163,E1 5.9786,E2 420.9894} C_DIS
LIN {X 115.6678,Y 69.968,Z 180,A 33.1643,B 5.8372,C 0.1594,E1 5.9761,E2 419.1858} C_DIS
LIN {X 113.3987,Y 73.5886,Z 180,A 34.9356,B 5.8374,C 0.1556,E1 5.9734,E2 417.4187} C_DIS
LIN {X 111.085,Y 77.0372,Z 180,A 36.6958,B 5.8374,C 0.1515,E1 5.9706,E2 415.6577} C_DIS
LIN {X 108.476,Y 80.6692,Z 180,A 38.4428,B 5.8375,C 0.1493,E1 5.9678,E2 413.9284} C_DIS
LIN {X 105.9176,Y 84.0004,Z 180,A 40.3165,B 5.8377,C 0.1439,E1 5.9646,E2 412.0426} C_DIS
LIN {X 102.6464,Y 87.968,Z 180,A 42.4709,B 5.8377,C 0.1395,E1 5.9607,E2 409.8906} C_DIS
LIN {X 99.604,Y 91.398,Z 180,A 44.278,B 5.8378,C 0.1374,E1 5.9573,E2 408.0998} C_DIS
LIN {X 95.6933,Y 95.4852,Z 180,A 46.7006,B 5.8379,C 0.1321,E1 5.9526,E2 405.6735} C_DIS
LIN {X 93.4069,Y 97.7226,Z 180,A 48.4998,B 5.8381,C 0.1229,E1 5.9489,E2 403.8194} C_DIS
LIN {X 89.9277,Y 100.934,Z 180,A 50.0135,B 5.8381,C 0.1263,E1 5.9459,E2 402.3661} C_DIS
LIN {X 86.6107,Y 103.7943,Z 180,A 51.9222,B 5.8381,C 0.1221,E1 5.9418,E2 400.4507} C_DIS
LIN {X 82.7817,Y 106.8726,Z 180,A 53.887,B 5.8381,C 0.1201,E1 5.9375,E2 398.5} C_DIS
LIN {X 79.1471,Y 109.5917,Z 180,A 55.775,B 5.8383,C 0.1173,E1 5.9333,E2 396.6163} C_DIS
LIN {X 75.5135,Y 112.1266,Z 180,A 57.5495,B 5.8383,C 0.1158,E1 5.9292,E2 394.8542} C_DIS
LIN {X 72.2724,Y 114.2422,Z 180,A 59.2264,B 5.8383,C 0.1127,E1 5.9252,E2 393.1729} C_DIS
LIN {X 68.7421,Y 116.4009,Z 180,A 60.9945,B 5.8383,C 0.1099,E1 5.921,E2 391.403} C_DIS
LIN {X 64.9863,Y 118.5387,Z 180,A 62.7946,B 5.8384,C 0.1077,E1 5.9166,E2 389.6067} C_DIS
LIN {X 61.5895,Y 120.3363,Z 180,A 64.2472,B 5.8384,C 0.108,E1 5.9131,E2 388.1755} C_DIS
LIN {X 58.4826,Y 121.8764,Z 180,A 65.6961,B 5.8384,C 0.1064,E1 5.9095,E2 386.7294} C_DIS
LIN {X 55.316,Y 123.3457,Z 180,A 67.2563,B 5.8385,C 0.1035,E1 5.9055,E2 385.1594} C_DIS
LIN {X 52.4511,Y 124.5915,Z 180,A 68.5715,B 5.8385,C 0.1021,E1 5.9021,E2 383.8455} C_DIS
LIN {X 49.5929,Y 125.7577,Z 180,A 69.9438,B 5.8385,C 0.0999,E1 5.8985,E2 382.4656} C_DIS
LIN {X 45.8922,Y 127.1532,Z 180,A 71.4665,B 5.8385,C 0.1002,E1 5.8946,E2 380.9618} C_DIS
LIN {X 42.9604,Y 128.1738,Z 180,A 72.8097,B 5.8385,C 0.0986,E1 5.891,E2 379.6155} C_DIS
LIN {X 36.5606,Y 130.1438,Z 180,A 75.4713,B 5.8386,C 0.0986,E1 5.884,E2 376.976} C_DIS
LIN {X 33.4526,Y 130.9772,Z 180,A 76.9937,B 5.8386,C 0.0954,E1 5.8798,E2 375.4347} C_DIS
LIN {X 29.9046,Y 131.8326,Z 180,A 78.5489,B 5.8386,C 0.0943,E1 5.8756,E2 373.8789} C_DIS
LIN {X 25.646,Y 132.727,Z 180,A 80.4494,B 5.8387,C 0.0925,E1 5.8703,E2 371.9721} C_DIS
LIN {X 21.6197,Y 133.4432,Z 180,A 82.1693,B 5.8387,C 0.0918,E1 5.8656,E2 370.2544} C_DIS
LIN {X 17.6431,Y 134.0255,Z 180,A 83.6576,B 5.8387,C 0.0938,E1 5.8616,E2 368.7927} C_DIS
LIN {X 10.5859,Y 134.7688,Z 180,A 86.8017,B 5.8387,C 0.0911,E1 5.8528,E2 365.6334} C_DIS
LIN {X 7.0475,Y 134.9983,Z 180,A 88.2851,B 5.8387,C 0.0911,E1 5.8486,E2 364.1529} C_DIS
LIN {X 3.6719,Y 135.1321,Z 180,A 89.9833,B 5.8387,C 0.0876,E1 5.8438,E2 362.4229} C_DIS
LIN {X 0.4375,Y 135.1816,Z 180,A 91.4472,B 5.8387,C 0.0864,E1 5.8397,E2 360.9483} C_DIS
LIN {X -3.2899,Y 135.1427,Z 180,A 92.7856,B 5.8387,C 0.0894,E1 5.836,E2 359.64} C_DIS
LIN {X -7.951,Y 134.9484,Z 180,A 94.6982,B 5.8387,C 0.0904,E1 5.8307,E2 357.7362} C_DIS
LIN {X -12.614,Y 134.5924,Z 180,A 97.0552,B 5.8387,C 0.0863,E1 5.8241,E2 355.3346} C_DIS
LIN {X -16.7079,Y 134.1471,Z 180,A 98.3415,B 5.8387,C 0.0924,E1 5.8206,E2 354.1051} C_DIS
LIN {X -20.6146,Y 133.6007,Z 180,A 100.0702,B 5.8387,C 0.0924,E1 5.8158,E2 352.3704} C_DIS
LIN {X -24.4611,Y 132.9518,Z 180,A 101.8353,B 5.8387,C 0.0918,E1 5.811,E2 350.5928} C_DIS
LIN {X -28.5224,Y 132.1384,Z 180,A 103.518,B 5.8387,C 0.0936,E1 5.8064,E2 348.9198} C_DIS
LIN {X -32.7228,Y 131.1625,Z 180,A 105.3635,B 5.8387,C 0.0946,E1 5.8014,E2 347.0733} C_DIS
LIN {X -36.171,Y 130.2528,Z 180,A 106.6816,B 5.8387,C 0.0979,E1 5.7979,E2 345.7795} C_DIS
LIN {X -38.9384,Y 129.4529,Z 180,A 108.2318,B 5.8387,C 0.0951,E1 5.7936,E2 344.1904} C_DIS
LIN {X -42.7106,Y 128.2569,Z 180,A 109.8515,B 5.8387,C 0.0972,E1 5.7893,E2 342.5786} C_DIS
LIN {X -49.7555,Y 125.6945,Z 180,A 113.0665,B 5.8386,C 0.0999,E1 5.7809,E2 339.3615} C_DIS
LIN {X -54.2544,Y 123.8181,Z 180,A 115.1144,B 5.8386,C 0.1023,E1 5.7757,E2 337.3172} C_DIS
LIN {X -57.978,Y 122.1174,Z 180,A 116.6679,B 5.8385,C 0.1064,E1 5.7718,E2 335.7869} C_DIS
LIN {X -61.1451,Y 120.5625,Z 180,A 118.1128,B 5.8385,C 0.1088,E1 5.7682,E2 334.3492} C_DIS
LIN {X -64.3926,Y 118.8622,Z 180,A 120.1075,B 5.8385,C 0.106,E1 5.7632,E2 332.3024} C_DIS
LIN {X -68.4129,Y 116.5943,Z 180,A 122.4372,B 5.8385,C 0.1048,E1 5.7574,E2 329.9287} C_DIS
LIN {X -72.4857,Y 114.1075,Z 180,A 124.1751,B 5.8384,C 0.1109,E1 5.7534,E2 328.2272} C_DIS
LIN {X -76.8504,Y 111.2148,Z 180,A 126.2926,B 5.8383,C 0.1155,E1 5.7485,E2 326.1238} C_DIS
LIN {X -80.4702,Y 108.6241,Z 180,A 128.1669,B 5.8383,C 0.1188,E1 5.7443,E2 324.2525} C_DIS
LIN {X -83.7885,Y 106.0856,Z 180,A 129.9856,B 5.8382,C 0.1213,E1 5.7403,E2 322.4295} C_DIS
LIN {X -87.1212,Y 103.366,Z 180,A 131.8064,B 5.8382,C 0.1247,E1 5.7364,E2 320.6105} C_DIS
LIN {X -90.3647,Y 100.5427,Z 180,A 133.629,B 5.838,C 0.1281,E1 5.7326,E2 318.7894} C_DIS
LIN {X -93.5868,Y 97.5506,Z 180,A 135.5311,B 5.838,C 0.1313,E1 5.7287,E2 316.8843} C_DIS
LIN {X -96.742,Y 94.4226,Z 180,A 137.496,B 5.8379,C 0.1343,E1 5.7248,E2 314.911} C_DIS
LIN {X -99.7418,Y 91.2481,Z 180,A 139.3815,B 5.8379,C 0.1378,E1 5.7212,E2 313.0229} C_DIS
LIN {X -102.7393,Y 87.8598,Z 180,A 141.3558,B 5.8377,C 0.1414,E1 5.7176,E2 311.0434} C_DIS
LIN {X -105.6333,Y 84.3576,Z 180,A 143.3104,B 5.8377,C 0.1453,E1 5.7142,E2 309.087} C_DIS
LIN {X -108.3888,Y 80.7862,Z 180,A 145.2232,B 5.8375,C 0.1497,E1 5.7109,E2 307.1757} C_DIS
LIN {X -110.9949,Y 77.1666,Z 180,A 147.1354,B 5.8375,C 0.1539,E1 5.7079,E2 305.2625} C_DIS
LIN {X -112.5902,Y 74.8203,Z 180,A 148.4241,B 5.8374,C 0.1559,E1 5.7059,E2 303.9644} C_DIS
LIN {X -115.5386,Y 70.1816,Z 180,A 150.8507,B 5.8372,C 0.1606,E1 5.7023,E2 301.5281} C_DIS
LIN {X -117.9139,Y 66.1127,Z 180,A 152.7775,B 5.8371,C 0.1662,E1 5.6996,E2 299.6116} C_DIS
LIN {X -119.391,Y 63.405,Z 180,A 154.6489,B 5.8371,C 0.164,E1 5.6971,E2 297.672} C_DIS
LIN {X -121.5636,Y 59.1342,Z 180,A 156.1743,B 5.8368,C 0.1741,E1 5.6953,E2 296.2107} C_DIS
LIN {X -123.2757,Y 55.4727,Z 180,A 157.7921,B 5.8367,C 0.1795,E1 5.6934,E2 294.6061} C_DIS
LIN {X -124.6419,Y 52.3306,Z 180,A 159.4268,B 5.8367,C 0.1816,E1 5.6916,E2 292.9503} C_DIS
LIN {X -125.9628,Y 49.0654,Z 180,A 160.8379,B 5.8365,C 0.1863,E1 5.6901,E2 291.5506} C_DIS
LIN {X -128.1736,Y 42.961,Z 180,A 163.5032,B 5.8362,C 0.1946,E1 5.6876,E2 288.8983} C_DIS
LIN {X -129.1903,Y 39.7992,Z 180,A 165.247,B 5.8362,C 0.1952,E1 5.6861,E2 287.1146} C_DIS
LIN {X -130.3002,Y 36.0014,Z 180,A 167.0454,B 5.8361,C 0.1987,E1 5.6848,E2 285.3028} C_DIS
LIN {X -131.5148,Y 31.2747,Z 180,A 169.042,B 5.8358,C 0.2051,E1 5.6834,E2 283.3168} C_DIS
LIN {X -132.4194,Y 27.1893,Z 180,A 170.8007,B 5.8357,C 0.2102,E1 5.6824,E2 281.5615} C_DIS
LIN {X -133.1018,Y 23.6228,Z 180,A 172.4384,B 5.8355,C 0.2136,E1 5.6816,E2 279.9129} C_DIS
LIN {X -133.7651,Y 19.5238,Z 180,A 174.2632,B 5.8354,C 0.2179,E1 5.6808,E2 278.0815} C_DIS
LIN {X -134.2524,Y 15.8255,Z 180,A 175.8255,B 5.8352,C 0.2226,E1 5.6802,E2 276.5229} C_DIS
LIN {X -134.6646,Y 11.8224,Z 180,A 177.6322,B 5.8351,C 0.2265,E1 5.6798,E2 274.7052} C_DIS
LIN {X -134.9471,Y 7.9714,Z 180,A 179.3672,B 5.8349,C 0.2302,E1 5.6794,E2 272.9593} C_DIS
LIN {X -135.1285,Y 3.8002,Z 180,A -178.9089,B 5.8347,C 0.2357,E1 5.6793,E2 271.2424} C_DIS
LIN {X -135.1835,Y -0.3568,Z 180,A -177.0693,B 5.8345,C 0.24,E1 5.6793,E2 269.3946} C_DIS
LIN {X -135.137,Y -3.4961,Z 180,A -175.7379,B 5.8344,C 0.2438,E1 5.6793,E2 268.0641} C_DIS
LIN {X -135.0169,Y -6.679,Z 180,A -174.3856,B 5.8342,C 0.2476,E1 5.6795,E2 266.7125} C_DIS
LIN {X -134.7913,Y -10.2781,Z 180,A -172.6739,B 5.8341,C 0.2502,E1 5.6798,E2 264.9792} C_DIS
LIN {X -134.4737,Y -13.8328,Z 180,A -171.191,B 5.8339,C 0.2548,E1 5.6802,E2 263.5012} C_DIS
LIN {X -134.0647,Y -17.3442,Z 180,A -169.6896,B 5.8337,C 0.259,E1 5.6808,E2 262.0005} C_DIS
LIN {X -133.4653,Y -21.4875,Z 180,A -167.8291,B 5.8335,C 0.2632,E1 5.6815,E2 260.1305} C_DIS
LIN {X -132.795,Y -25.2901,Z 180,A -166.1795,B 5.8333,C 0.2676,E1 5.6824,E2 258.4804} C_DIS
LIN {X -131.9729,Y -29.2891,Z 180,A -164.4664,B 5.8331,C 0.2726,E1 5.6834,E2 256.7707} C_DIS
LIN {X -131.0029,Y -33.3516,Z 180,A -162.4462,B 5.833,C 0.275,E1 5.6847,E2 254.7203} C_DIS
LIN {X -129.7834,Y -37.82,Z 180,A -160.5953,B 5.8327,C 0.2815,E1 5.6861,E2 252.8847} C_DIS
LIN {X -128.6645,Y -41.4683,Z 180,A -158.9298,B 5.8325,C 0.2854,E1 5.6875,E2 251.2142} C_DIS
LIN {X -127.3687,Y -45.2944,Z 180,A -156.7499,B 5.8325,C 0.2854,E1 5.6896,E2 248.9766} C_DIS
LIN {X -125.9688,Y -49.0499,Z 180,A -155.4593,B 5.8321,C 0.2939,E1 5.6909,E2 247.7382} C_DIS
LIN {X -124.5773,Y -52.4853,Z 180,A -153.758,B 5.8319,C 0.2967,E1 5.6927,E2 246.0215} C_DIS
LIN {X -122.8233,Y -56.467,Z 180,A -152.0019,B 5.8316,C 0.3023,E1 5.6947,E2 244.2774} C_DIS
LIN {X -121.1622,Y -59.9478,Z 180,A -150.3318,B 5.8314,C 0.3061,E1 5.6967,E2 242.6037} C_DIS
LIN {X -119.8516,Y -62.5277,Z 180,A -148.5933,B 5.8315,C 0.304,E1 5.6991,E2 240.8013} C_DIS
LIN {X -117.8614,Y -66.2058,Z 180,A -146.9578,B 5.8312,C 0.3097,E1 5.7013,E2 239.184} C_DIS
LIN {X -116.2596,Y -68.9806,Z 180,A -145.7339,B 5.831,C 0.3144,E1 5.703,E2 237.9776} C_DIS
LIN {X -113.8564,Y -72.8785,Z 180,A -143.7873,B 5.8307,C 0.3189,E1 5.7059,E2 236.031} C_DIS
LIN {X -111.7068,Y -76.1336,Z 180,A -142.0515,B 5.8306,C 0.3219,E1 5.7086,E2 234.2856} C_DIS
LIN {X -109.1222,Y -79.7933,Z 180,A -140.1191,B 5.8304,C 0.3258,E1 5.7117,E2 232.3496} C_DIS
LIN {X -106.3137,Y -83.4982,Z 180,A -138.1482,B 5.8301,C 0.3302,E1 5.7151,E2 230.3794} C_DIS
LIN {X -103.438,Y -87.0354,Z 180,A -136.1877,B 5.8299,C 0.334,E1 5.7186,E2 228.4158} C_DIS
LIN {X -101.0684,Y -89.7765,Z 180,A -134.3828,B 5.8299,C 0.3343,E1 5.722,E2 226.5773} C_DIS
LIN {X -98.8094,Y -92.2566,Z 180,A -133.1499,B 5.8296,C 0.3392,E1 5.7243,E2 225.3687} C_DIS
LIN {X -95.7085,Y -95.4699,Z 180,A -131.244,B 5.8294,C 0.3428,E1 5.728,E2 223.4616} C_DIS
LIN {X -92.4576,Y -98.6221,Z 180,A -129.2629,B 5.8292,C 0.3458,E1 5.7321,E2 221.4731} C_DIS
LIN {X -89.1249,Y -101.6435,Z 180,A -127.2539,B 5.8291,C 0.3481,E1 5.7363,E2 219.4514} C_DIS
LIN {X -85.3704,Y -104.8165,Z 180,A -125.2743,B 5.8288,C 0.3529,E1 5.7405,E2 217.4853} C_DIS
LIN {X -81.9285,Y -107.5283,Z 180,A -123.3937,B 5.8286,C 0.3557,E1 5.7447,E2 215.6019} C_DIS
LIN {X -78.5535,Y -110.0177,Z 180,A -121.5652,B 5.8285,C 0.358,E1 5.7488,E2 213.7671} C_DIS
LIN {X -74.9377,Y -112.5118,Z 180,A -119.6568,B 5.8283,C 0.3602,E1 5.7532,E2 211.8528} C_DIS
LIN {X -71.1273,Y -114.9591,Z 180,A -117.6922,B 5.8283,C 0.3625,E1 5.7579,E2 209.8826} C_DIS
LIN {X -67.2835,Y -117.2502,Z 180,A -115.7611,B 5.8281,C 0.3646,E1 5.7626,E2 207.947} C_DIS
LIN {X -63.4486,Y -119.368,Z 180,A -113.9442,B 5.8279,C 0.3674,E1 5.767,E2 206.1351} C_DIS
LIN {X -60.1768,Y -121.0493,Z 180,A -112.395,B 5.8278,C 0.3694,E1 5.7709,E2 204.5871} C_DIS
LIN {X -57.2565,Y -122.4583,Z 180,A -111.0002,B 5.8277,C 0.3707,E1 5.7744,E2 203.1895} C_DIS
LIN {X -53.7566,Y -124.0333,Z 180,A -109.4809,B 5.8275,C 0.3736,E1 5.7782,E2 201.6838} C_DIS
LIN {X -50.7724,Y -125.2847,Z 180,A -107.9181,B 5.8275,C 0.3727,E1 5.7823,E2 200.0963} C_DIS
LIN {X -46.465,Y -126.9467,Z 180,A -105.927,B 5.8275,C 0.374,E1 5.7876,E2 198.1006} C_DIS
LIN {X -39.7395,Y -129.2085,Z 180,A -103.1718,B 5.8271,C 0.3794,E1 5.7948,E2 195.3771} C_DIS
LIN {X -36.6438,Y -130.1205,Z 180,A -101.6804,B 5.8271,C 0.3788,E1 5.7988,E2 193.8696} C_DIS
LIN {X -33.9269,Y -130.8568,Z 180,A -100.3564,B 5.8272,C 0.378,E1 5.8025,E2 192.5286} C_DIS
LIN {X -30.0608,Y -131.7969,Z 180,A -98.7595,B 5.8271,C 0.38,E1 5.8068,E2 190.9427} C_DIS
LIN {X -26.1735,Y -132.6261,Z 180,A -96.9213,B 5.8271,C 0.3788,E1 5.8118,E2 189.0844} C_DIS
LIN {X -22.7823,Y -133.2493,Z 180,A -95.5197,B 5.8271,C 0.3801,E1 5.8157,E2 187.6899} C_DIS
LIN {X -19.1621,Y -133.8168,Z 180,A -93.3278,B 5.8276,C 0.3724,E1 5.822,E2 185.4152} C_DIS
LIN {X -13.6402,Y -134.4939,Z 180,A -91.7168,B 5.8269,C 0.3825,E1 5.8262,E2 183.8997} C_DIS
LIN {X -9.9682,Y -134.8139,Z 180,A -90.0609,B 5.827,C 0.3814,E1 5.8308,E2 182.231} C_DIS
LIN {X -6.113,Y -135.0453,Z 180,A -88.3019,B 5.8271,C 0.3799,E1 5.8358,E2 180.4557} C_DIS
LIN {X 0.9555,Y -135.1708,Z 180,A -86.5836,B 5.826,C 0.3963,E1 5.8402,E2 178.8986} C_DIS
Enddeposition()
LIN {X 0.9555,Y -135.1708,Z 180,A -86.5838,B 5.826,C 0.3963,E1 5.8402,E2 178.8989} C_DIS
Startdeposition()
$VEL.CP = VEL_PRINT
LIN {X -0.5442,Y -136.0837,Z 180,A -87.1958,B 5.5803,C 0.3963,E1 5.5929,E2 179.6128} C_DIS
LIN {X -5.4533,Y -135.9754,Z 180,A -89.3253,B 5.5803,C 0.3971,E1 5.587,E2 181.7511} C_DIS
LIN {X -10.773,Y -135.6592,Z 180,A -91.0086,B 5.5807,C 0.39,E1 5.5825,E2 183.3641} C_DIS
LIN {X -16.3731,Y -135.096,Z 180,A -93.5623,B 5.5807,C 0.3918,E1 5.5753,E2 185.9421} C_DIS
LIN {X -19.5696,Y -134.6704,Z 180,A -94.6201,B 5.5809,C 0.3878,E1 5.5725,E2 186.9622} C_DIS
LIN {X -22.0869,Y -134.2804,Z 180,A -95.7797,B 5.5809,C 0.3885,E1 5.5693,E2 188.1333} C_DIS
LIN {X -25.5425,Y -133.6658,Z 180,A -97.1639,B 5.5809,C 0.3868,E1 5.5655,E2 189.506} C_DIS
LIN {X -28.5923,Y -133.0468,Z 180,A -98.5215,B 5.5809,C 0.3868,E1 5.5617,E2 190.87} C_DIS
LIN {X -32.0036,Y -132.2676,Z 180,A -99.9799,B 5.581,C 0.3858,E1 5.5578,E2 192.3269} C_DIS
LIN {X -35.3594,Y -131.4106,Z 180,A -101.455,B 5.581,C 0.3851,E1 5.5538,E2 193.8046} C_DIS
LIN {X -39.2127,Y -130.3138,Z 180,A -103.7255,B 5.5807,C 0.3907,E1 5.5475,E2 196.1496} C_DIS
LIN {X -43.7254,Y -128.8705,Z 180,A -105.1462,B 5.5813,C 0.3826,E1 5.5439,E2 197.4979} C_DIS
LIN {X -46.3965,Y -127.9309,Z 180,A -106.3753,B 5.5813,C 0.382,E1 5.5407,E2 198.7319} C_DIS
LIN {X -50.0566,Y -126.5459,Z 180,A -108.0271,B 5.5813,C 0.3805,E1 5.5364,E2 200.3845} C_DIS
LIN {X -52.8678,Y -125.3957,Z 180,A -109.3049,B 5.5815,C 0.3793,E1 5.5331,E2 201.6624} C_DIS
LIN {X -56.3661,Y -123.8645,Z 180,A -110.9371,B 5.5815,C 0.3779,E1 5.5289,E2 203.2979} C_DIS
LIN {X -59.2845,Y -122.4936,Z 180,A -112.311,B 5.5817,C 0.3765,E1 5.5254,E2 204.674} C_DIS
LIN {X -62.1783,Y -121.0494,Z 180,A -113.7344,B 5.5817,C 0.3756,E1 5.5219,E2 206.1052} C_DIS
LIN {X -65.8714,Y -119.0814,Z 180,A -115.5719,B 5.5818,C 0.3742,E1 5.5173,E2 207.9525} C_DIS
LIN {X -69.855,Y -116.7893,Z 180,A -117.5267,B 5.582,C 0.3718,E1 5.5126,E2 209.9098} C_DIS
LIN {X -73.2761,Y -114.6737,Z 180,A -119.1906,B 5.5822,C 0.3691,E1 5.5087,E2 211.5699} C_DIS
LIN {X -76.8425,Y -112.3151,Z 180,A -121.107,B 5.5822,C 0.3676,E1 5.5042,E2 213.501} C_DIS
LIN {X -80.7793,Y -109.518,Z 180,A -123.1077,B 5.5825,C 0.3641,E1 5.4997,E2 215.4974} C_DIS
LIN {X -84.2182,Y -106.896,Z 180,A -124.9703,B 5.5827,C 0.3615,E1 5.4956,E2 217.3651} C_DIS
LIN {X -87.6445,Y -104.1053,Z 180,A -126.9112,B 5.5828,C 0.3591,E1 5.4914,E2 219.3159} C_DIS
LIN {X -90.898,Y -101.2768,Z 180,A -128.7073,B 5.583,C 0.3556,E1 5.4876,E2 221.1093} C_DIS
LIN {X -94.1687,Y -98.2431,Z 180,A -130.637,B 5.5832,C 0.3526,E1 5.4837,E2 223.0451} C_DIS
LIN {X -96.9741,Y -95.4752,Z 180,A -132.3466,B 5.5834,C 0.3499,E1 5.4803,E2 224.7608} C_DIS
LIN {X -100.7537,Y -91.4773,Z 180,A -134.5916,B 5.5837,C 0.3445,E1 5.4761,E2 226.9962} C_DIS
LIN {X -103.3664,Y -88.5153,Z 180,A -136.4098,B 5.5838,C 0.3426,E1 5.4727,E2 228.8335} C_DIS
LIN {X -106.214,Y -85.0775,Z 180,A -138.3155,B 5.5841,C 0.3388,E1 5.4693,E2 230.7419} C_DIS
LIN {X -108.9267,Y -81.5753,Z 180,A -140.1704,B 5.5843,C 0.3346,E1 5.4662,E2 232.5949} C_DIS
LIN {X -111.4502,Y -78.0926,Z 180,A -142.0812,B 5.5845,C 0.3315,E1 5.4631,E2 234.5176} C_DIS
LIN {X -114.0552,Y -74.2351,Z 180,A -144.0249,B 5.5848,C 0.3268,E1 5.4601,E2 236.4585} C_DIS
LIN {X -116.2129,Y -70.8108,Z 180,A -145.8159,B 5.585,C 0.3236,E1 5.4574,E2 238.2597} C_DIS
LIN {X -119.7988,Y -64.5578,Z 180,A -148.8389,B 5.5854,C 0.3161,E1 5.4533,E2 241.2798} C_DIS
LIN {X -121.4171,Y -61.456,Z 180,A -150.3433,B 5.5856,C 0.3127,E1 5.4514,E2 242.7874} C_DIS
LIN {X -123.2713,Y -57.6489,Z 180,A -152.0305,B 5.5859,C 0.3072,E1 5.4493,E2 244.4617} C_DIS
LIN {X -124.5084,Y -54.9274,Z 180,A -153.4002,B 5.586,C 0.3051,E1 5.4477,E2 245.8448} C_DIS
LIN {X -125.6996,Y -52.1402,Z 180,A -154.7425,B 5.5862,C 0.3024,E1 5.4463,E2 247.1946} C_DIS
LIN {X -127.1458,Y -48.5133,Z 180,A -156.8034,B 5.5862,C 0.3019,E1 5.4442,E2 249.3066} C_DIS
LIN {X -128.3936,Y -45.1031,Z 180,A -158.1543,B 5.5865,C 0.2962,E1 5.4429,E2 250.6345} C_DIS
LIN {X -129.7415,Y -41.0633,Z 180,A -160.0758,B 5.5867,C 0.2925,E1 5.4413,E2 252.5708} C_DIS
LIN {X -131.1142,Y -36.4424,Z 180,A -162.5577,B 5.5867,C 0.2911,E1 5.4394,E2 255.1074} C_DIS
LIN {X -132.4006,Y -31.4518,Z 180,A -164.1206,B 5.5873,C 0.2796,E1 5.4384,E2 256.5939} C_DIS
LIN {X -133.2846,Y -27.4644,Z 180,A -165.9392,B 5.5875,C 0.2758,E1 5.4373,E2 258.4237} C_DIS
LIN {X -134.0231,Y -23.5989,Z 180,A -167.5423,B 5.5878,C 0.2707,E1 5.4365,E2 260.0189} C_DIS
LIN {X -134.5525,Y -20.3665,Z 180,A -169.0362,B 5.5879,C 0.2678,E1 5.4358,E2 261.5262} C_DIS
LIN {X -135.1078,Y -16.2753,Z 180,A -170.7958,B 5.5881,C 0.2631,E1 5.4352,E2 263.2871} C_DIS
LIN {X -135.5267,Y -12.3275,Z 180,A -172.6587,B 5.5883,C 0.2601,E1 5.4347,E2 265.1726} C_DIS
LIN {X -135.8364,Y -8.2169,Z 180,A -174.2663,B 5.5886,C 0.254,E1 5.4344,E2 266.763} C_DIS
LIN {X -136.0058,Y -4.6725,Z 180,A -175.9527,B 5.5886,C 0.2515,E1 5.4342,E2 268.4721} C_DIS
LIN {X -136.0858,Y -0.4091,Z 180,A -177.6436,B 5.5889,C 0.2455,E1 5.4342,E2 270.1488} C_DIS
LIN {X -136.0421,Y 3.4215,Z 180,A -179.3665,B 5.5891,C 0.2418,E1 5.4342,E2 271.884} C_DIS
LIN {X -135.9049,Y 6.9922,Z 180,A 179.153,B 5.5893,C 0.2373,E1 5.4344,E2 273.3603} C_DIS
LIN {X -135.6658,Y 10.6946,Z 180,A 177.3943,B 5.5894,C 0.2346,E1 5.4347,E2 275.142} C_DIS
LIN {X -135.3037,Y 14.5564,Z 180,A 175.7926,B 5.5896,C 0.2297,E1 5.4352,E2 276.7385} C_DIS
LIN {X -134.7791,Y 18.809,Z 180,A 173.9382,B 5.5898,C 0.2251,E1 5.4359,E2 278.5976} C_DIS
LIN {X -134.1785,Y 22.6976,Z 180,A 172.2795,B 5.59,C 0.2204,E1 5.4366,E2 280.2552} C_DIS
LIN {X -133.4139,Y 26.8285,Z 180,A 170.4578,B 5.5902,C 0.2159,E1 5.4376,E2 282.0819} C_DIS
LIN {X -132.6472,Y 30.3918,Z 180,A 168.8842,B 5.5903,C 0.212,E1 5.4385,E2 283.659} C_DIS
LIN {X -131.8017,Y 33.8736,Z 180,A 167.0404,B 5.5903,C 0.2108,E1 5.4398,E2 285.5425} C_DIS
LIN {X -130.9159,Y 37.1514,Z 180,A 165.7644,B 5.5905,C 0.2055,E1 5.4408,E2 286.7986} C_DIS
LIN {X -129.702,Y 41.1867,Z 180,A 163.8898,B 5.5907,C 0.2016,E1 5.4423,E2 288.6839} C_DIS
LIN {X -127.6789,Y 47.09,Z 180,A 161.445,B 5.591,C 0.1929,E1 5.4446,E2 291.1041} C_DIS
LIN {X -126.7413,Y 49.554,Z 180,A 160.2457,B 5.591,C 0.1907,E1 5.4458,E2 292.3134} C_DIS
LIN {X -125.4607,Y 52.7123,Z 180,A 158.7674,B 5.5912,C 0.1873,E1 5.4473,E2 293.7956} C_DIS
LIN {X -124.0641,Y 55.9207,Z 180,A 157.2479,B 5.5912,C 0.1839,E1 5.4491,E2 295.3195} C_DIS
LIN {X -122.2687,Y 59.7453,Z 180,A 154.5256,B 5.5912,C 0.1878,E1 5.4526,E2 298.1542} C_DIS
LIN {X -119.2658,Y 65.5381,Z 180,A 152.8072,B 5.5917,C 0.1716,E1 5.4546,E2 299.746} C_DIS
LIN {X -116.3773,Y 70.5391,Z 180,A 150.3022,B 5.5918,C 0.1663,E1 5.4582,E2 302.2579} C_DIS
LIN {X -113.4351,Y 75.1803,Z 180,A 147.8508,B 5.592,C 0.162,E1 5.4619,E2 304.7242} C_DIS
LIN {X -111.605,Y 77.8702,Z 180,A 146.2919,B 5.592,C 0.1606,E1 5.4644,E2 306.3048} C_DIS
LIN {X -108.9922,Y 81.4873,Z 180,A 144.3773,B 5.5921,C 0.1566,E1 5.4675,E2 308.2221} C_DIS
LIN {X -106.6241,Y 84.5623,Z 180,A 142.6894,B 5.5922,C 0.1534,E1 5.4705,E2 309.9151} C_DIS
LIN {X -103.8183,Y 87.9842,Z 180,A 140.7708,B 5.5923,C 0.1499,E1 5.4739,E2 311.8389} C_DIS
LIN {X -100.9058,Y 91.3097,Z 180,A 138.8791,B 5.5924,C 0.1462,E1 5.4774,E2 313.7326} C_DIS
LIN {X -97.7342,Y 94.6966,Z 180,A 136.9226,B 5.5925,C 0.1422,E1 5.4812,E2 315.6878} C_DIS
LIN {X -94.5308,Y 97.8947,Z 180,A 134.977,B 5.5925,C 0.1388,E1 5.4851,E2 317.6366} C_DIS
LIN {X -91.2005,Y 101.0049,Z 180,A 133.018,B 5.5927,C 0.1355,E1 5.4891,E2 319.5989} C_DIS
LIN {X -87.8987,Y 103.891,Z 180,A 131.1191,B 5.5927,C 0.1326,E1 5.4931,E2 321.5026} C_DIS
LIN {X -84.4131,Y 106.7428,Z 180,A 129.165,B 5.5928,C 0.1299,E1 5.4974,E2 323.4621} C_DIS
LIN {X -80.8078,Y 109.497,Z 180,A 127.2324,B 5.5928,C 0.1268,E1 5.5017,E2 325.3959} C_DIS
LIN {X -77.0503,Y 112.1725,Z 180,A 125.2946,B 5.5929,C 0.1237,E1 5.5061,E2 327.3316} C_DIS
LIN {X -70.0416,Y 116.6781,Z 180,A 121.8263,B 5.5931,C 0.118,E1 5.5143,E2 330.7924} C_DIS
LIN {X -66.6462,Y 118.6495,Z 180,A 120.0567,B 5.5931,C 0.1169,E1 5.5186,E2 332.5747} C_DIS
LIN {X -63.1128,Y 120.5639,Z 180,A 118.385,B 5.5931,C 0.1144,E1 5.5227,E2 334.2428} C_DIS
LIN {X -59.5017,Y 122.3888,Z 180,A 116.726,B 5.5931,C 0.1119,E1 5.5269,E2 335.8951} C_DIS
LIN {X -56.4698,Y 123.8166,Z 180,A 115.2016,B 5.5932,C 0.1114,E1 5.5308,E2 337.4322} C_DIS
LIN {X -51.9953,Y 125.7601,Z 180,A 113.2081,B 5.5932,C 0.1085,E1 5.5359,E2 339.4169} C_DIS
LIN {X -48.0789,Y 127.3085,Z 180,A 110.7782,B 5.5932,C 0.1138,E1 5.5424,E2 341.9242} C_DIS
LIN {X -43.2626,Y 129.0245,Z 180,A 109.4715,B 5.5934,C 0.1027,E1 5.5456,E2 343.1281} C_DIS
LIN {X -38.9314,Y 130.3986,Z 180,A 107.1348,B 5.5934,C 0.1058,E1 5.552,E2 345.5147} C_DIS
LIN {X -34.5476,Y 131.627,Z 180,A 105.2524,B 5.5934,C 0.1041,E1 5.557,E2 347.3918} C_DIS
LIN {X -30.3086,Y 132.6662,Z 180,A 103.5035,B 5.5934,C 0.1019,E1 5.5617,E2 349.1288} C_DIS
LIN {X -26.7609,Y 133.4277,Z 180,A 101.8814,B 5.5934,C 0.1022,E1 5.5662,E2 350.7614} C_DIS
LIN {X -22.5766,Y 134.1987,Z 180,A 100.149,B 5.5934,C 0.1007,E1 5.5709,E2 352.4857} C_DIS
LIN {X -18.448,Y 134.8304,Z 180,A 98.3519,B 5.5934,C 0.1005,E1 5.5759,E2 354.2866} C_DIS
LIN {X -10.8498,Y 135.6527,Z 180,A 94.8228,B 5.5934,C 0.1033,E1 5.5858,E2 357.8513} C_DIS
LIN {X -7.0886,Y 135.9001,Z 180,A 93.8606,B 5.5934,C 0.0958,E1 5.5883,E2 358.7377} C_DIS
LIN {X -4.1077,Y 136.023,Z 180,A 91.6596,B 5.5933,C 0.1068,E1 5.5948,E2 361.0513} C_DIS
LIN {X 1.4597,Y 136.0778,Z 180,A 90.0011,B 5.5934,C 0.0988,E1 5.5992,E2 362.6269} C_DIS
LIN {X 6.1219,Y 135.9486,Z 180,A 88.1422,B 5.5934,C 0.0978,E1 5.6043,E2 364.4724} C_DIS
LIN {X 10.2525,Y 135.6982,Z 180,A 85.8869,B 5.5934,C 0.1044,E1 5.6108,E2 366.7886} C_DIS
LIN {X 14.3188,Y 135.3293,Z 180,A 84.6259,B 5.5934,C 0.0994,E1 5.6141,E2 367.994} C_DIS
LIN {X 17.6544,Y 134.9344,Z 180,A 83.2093,B 5.5934,C 0.1,E1 5.6181,E2 369.4104} C_DIS
LIN {X 21.1213,Y 134.4357,Z 180,A 81.7431,B 5.5934,C 0.1006,E1 5.6221,E2 370.8751} C_DIS
LIN {X 25.2436,Y 133.7229,Z 180,A 79.9612,B 5.5934,C 0.1018,E1 5.627,E2 372.6589} C_DIS
LIN {X 28.757,Y 133.0112,Z 180,A 78.4637,B 5.5934,C 0.1025,E1 5.6311,E2 374.1546} C_DIS
LIN {X 32.3998,Y 132.1721,Z 180,A 76.9413,B 5.5934,C 0.103,E1 5.6352,E2 375.6704} C_DIS
LIN {X 36.015,Y 131.2337,Z 180,A 74.7987,B 5.5932,C 0.1114,E1 5.6412,E2 377.8812} C_DIS
LIN {X 40.5991,Y 129.8894,Z 180,A 73.3895,B 5.5933,C 0.1055,E1 5.6448,E2 379.2176} C_DIS
LIN {X 44.8984,Y 128.4646,Z 180,A 71.4257,B 5.5933,C 0.108,E1 5.65,E2 381.1879} C_DIS
LIN {X 48.7823,Y 127.0413,Z 180,A 69.6297,B 5.5933,C 0.1105,E1 5.6547,E2 382.9902} C_DIS
LIN {X 52.3322,Y 125.6194,Z 180,A 68.0924,B 5.5933,C 0.1114,E1 5.6586,E2 384.5186} C_DIS
LIN {X 56.2728,Y 123.9066,Z 180,A 66.38,B 5.5932,C 0.1122,E1 5.663,E2 386.2191} C_DIS
LIN {X 59.0118,Y 122.6239,Z 180,A 65.119,B 5.5932,C 0.1137,E1 5.6661,E2 387.4784} C_DIS
LIN {X 62.1621,Y 121.0577,Z 180,A 63.6423,B 5.5932,C 0.1155,E1 5.6698,E2 388.9546} C_DIS
LIN {X 65.5132,Y 119.2795,Z 180,A 61.9522,B 5.593,C 0.119,E1 5.674,E2 390.6559} C_DIS
LIN {X 69.4576,Y 117.0262,Z 180,A 60.0591,B 5.593,C 0.1215,E1 5.6786,E2 392.5467} C_DIS
LIN {X 73.3989,Y 114.595,Z 180,A 58.2101,B 5.593,C 0.1231,E1 5.6829,E2 394.3835} C_DIS
LIN {X 76.8425,Y 112.3151,Z 180,A 56.4357,B 5.5929,C 0.1264,E1 5.687,E2 396.1623} C_DIS
LIN {X 80.3949,Y 109.8004,Z 180,A 54.6363,B 5.5929,C 0.1291,E1 5.6911,E2 397.9579} C_DIS
LIN {X 84.0083,Y 107.0608,Z 180,A 52.8242,B 5.5928,C 0.1311,E1 5.6951,E2 399.7583} C_DIS
LIN {X 86.968,Y 104.6711,Z 180,A 51.3292,B 5.5928,C 0.1325,E1 5.6983,E2 401.2406} C_DIS
LIN {X 89.7693,Y 102.2793,Z 180,A 49.6829,B 5.5926,C 0.1367,E1 5.7018,E2 402.8988} C_DIS
LIN {X 95.6929,Y 96.7594,Z 180,A 46.6088,B 5.5926,C 0.1387,E1 5.708,E2 405.9327} C_DIS
LIN {X 99.5514,Y 92.7844,Z 180,A 44.018,B 5.5924,C 0.1472,E1 5.7131,E2 408.5558} C_DIS
LIN {X 102.67,Y 89.3215,Z 180,A 42.1259,B 5.5923,C 0.1504,E1 5.7165,E2 410.4398} C_DIS
LIN {X 105.5483,Y 85.9013,Z 180,A 40.2828,B 5.5922,C 0.154,E1 5.7198,E2 412.2787} C_DIS
LIN {X 108.1968,Y 82.5402,Z 180,A 38.7288,B 5.5922,C 0.1545,E1 5.7224,E2 413.803} C_DIS
LIN {X 110.0022,Y 80.1189,Z 180,A 37.2283,B 5.592,C 0.1607,E1 5.725,E2 415.332} C_DIS
LIN {X 112.5465,Y 76.5035,Z 180,A 35.4149,B 5.5919,C 0.1644,E1 5.7278,E2 417.1402} C_DIS
LIN {X 115.0833,Y 72.631,Z 180,A 33.5036,B 5.5918,C 0.1685,E1 5.7307,E2 419.0477} C_DIS
LIN {X 117.5316,Y 68.5995,Z 180,A 31.575,B 5.5917,C 0.1725,E1 5.7335,E2 420.9701} C_DIS
LIN {X 119.6697,Y 64.7979,Z 180,A 29.7554,B 5.5915,C 0.1769,E1 5.7359,E2 422.7884} C_DIS
LIN {X 121.514,Y 61.2657,Z 180,A 28.244,B 5.5915,C 0.1787,E1 5.7378,E2 424.2801} C_DIS
LIN {X 122.9382,Y 58.3539,Z 180,A 26.826,B 5.5913,C 0.183,E1 5.7396,E2 425.7053} C_DIS
LIN {X 124.632,Y 54.6464,Z 180,A 24.6614,B 5.591,C 0.1941,E1 5.7421,E2 427.9259} C_DIS
LIN {X 126.4721,Y 50.241,Z 180,A 23.2975,B 5.591,C 0.1898,E1 5.7434,E2 429.2115} C_DIS
LIN {X 127.5669,Y 47.389,Z 180,A 22.0277,B 5.591,C 0.1929,E1 5.7447,E2 430.48} C_DIS
LIN {X 128.7448,Y 44.0903,Z 180,A 20.4337,B 5.5908,C 0.1987,E1 5.7461,E2 432.0895} C_DIS
LIN {X 130.1336,Y 39.8016,Z 180,A 18.7192,B 5.5908,C 0.2011,E1 5.7476,E2 433.7824} C_DIS
LIN {X 131.2316,Y 36.0225,Z 180,A 17.1233,B 5.5906,C 0.2047,E1 5.7488,E2 435.3718} C_DIS
LIN {X 131.9237,Y 33.3928,Z 180,A 15.9633,B 5.5904,C 0.2081,E1 5.7496,E2 436.5344} C_DIS
LIN {X 132.866,Y 29.4294,Z 180,A 14.1993,B 5.5902,C 0.2136,E1 5.7507,E2 438.3056} C_DIS
LIN {X 133.6393,Y 25.681,Z 180,A 12.7292,B 5.5902,C 0.2159,E1 5.7515,E2 439.7592} C_DIS
LIN {X 134.2415,Y 22.3202,Z 180,A 11.3281,B 5.59,C 0.2194,E1 5.7522,E2 441.1566} C_DIS
LIN {X 134.8263,Y 18.4787,Z 180,A 9.5842,B 5.5898,C 0.2257,E1 5.7529,E2 442.9152} C_DIS
LIN {X 135.3408,Y 14.2122,Z 180,A 7.9318,B 5.5897,C 0.2284,E1 5.7534,E2 444.5493} C_DIS
LIN {X 135.7235,Y 9.9058,Z 180,A 5.6063,B 5.5891,C 0.2413,E1 5.7539,E2 446.9389} C_DIS
LIN {X 135.9961,Y 4.9233,Z 180,A 3.3431,B 5.5887,C 0.2497,E1 5.7541,E2 449.2236} C_DIS
LIN {X 136.0802,Y -1.2484,Z 180,A 1.5942,B 5.589,C 0.2442,E1 5.7541,E2 450.8691} C_DIS
LIN {X 135.8039,Y -8.7444,Z 180,A -1.862,B 5.5884,C 0.2578,E1 5.7536,E2 454.365} C_DIS
LIN {X 135.4971,Y -12.6359,Z 180,A -2.8876,B 5.5886,C 0.253,E1 5.7534,E2 455.3146} C_DIS
LIN {X 135.0148,Y -17.0412,Z 180,A -4.9454,B 5.5882,C 0.2612,E1 5.7527,E2 457.3981} C_DIS
LIN {X 134.1133,Y -23.0835,Z 180,A -7.332,B 5.588,C 0.2657,E1 5.7517,E2 459.7635} C_DIS
Enddeposition()
END
